// TwinCAT 3 PLC project XtsTransport
// Title: XTS Transport
// Author: D.Hauer
// ProjectVersion: 3.2.8
// Description: basic functionblocks for building XTS transport
// ProgramVersion: 3.1.4026.19
// libraries:
//   Tc2_Math, * (Beckhoff Automation GmbH)
//   Tc2_MC2, * (Beckhoff Automation GmbH)
//   Tc2_Standard, * (Beckhoff Automation GmbH)
//   Tc2_System, * (Beckhoff Automation GmbH)
//   Tc2_Utilities, * (Beckhoff Automation GmbH)
//   Tc3_McCollisionAvoidance, * (Beckhoff Automation GmbH)
//   Tc3_McCoordinatedMotion, * (Beckhoff Automation GmbH)
//   Tc3_Module, * (Beckhoff Automation GmbH)
//   Tc3_XTS_Utility, * (Beckhoff Automation GmbH)
//   VisuDialogs, * (System)
// project tree:
//   / GlobalTextList.TcGTLO (not stored), MAIN.TcPOU, PlcTask.TcTTO
//   MAPPING/ MAPPING_in.TcPOU, MAPPING_out.TcPOU
//   MAPPING/_types/ U_GEAR_DATA.TcDUT (not stored), U_MOVER_CTRL.TcDUT (not stored), U_MOVER_INFO.TcDUT (not stored), U_MOVER_STATE.TcDUT (not stored), U_MOVE_DATA.TcDUT (not stored), U_XTS_STATION_CTRL.TcDUT (not stored), U_XTS_STATION_STATE.TcDUT (not stored), U_XTS_TRANSPORT_CTRL.TcDUT (not stored), U_XTS_TRANSPORT_STATE.TcDUT (not stored)
//   MSG/ fb_LocalTime.TcPOU (not stored), f_MessageSet.TcPOU, GVL_MSG.TcGVL, MessageData.TcPOU (not stored), T_MESSAGE_LIST.TcVIS
//   MSG/types/ e_Device.TcDUT (not stored), E_MessageType.TcDUT (not stored), E_MESSAGE_STATE.TcDUT, e_Subdevice.TcDUT (not stored), ST_Message.TcDUT (not stored), TL_E_MESSAGETYPE.TcTLO
//   XTS/CaGroup/ FB_CaGroup.TcPOU, I_XtsTransport_CaGroup.TcIO (not stored)
//   XTS/CaGroup/types/ E_CA_GROUP_STATE.TcDUT (not stored), E_GROUP_CHECK.TcDUT (not stored), ST_GROUP_INFO.TcDUT (not stored)
//   XTS/ GVL_XTS.TcGVL (not stored), XTS_Parameter.TcGVL
//   XTS/Mover/ fb_Mover.TcPOU, fb_MoverCtrl.TcPOU (not stored), I_XtsTransport_Mover.TcIO
//   XTS/Mover/types/ E_MOVER_CTRL.TcDUT (not stored), E_MOVER_STATE.TcDUT, ST_GEAR_DATA.TcDUT, ST_MOVER_CTRL.TcDUT (not stored), ST_MOVER_INFO.TcDUT (not stored), ST_MOVER_STATE.TcDUT (not stored), ST_MOVE_DATA.TcDUT (not stored)
//   XTS/XtsStation/ fb_Station.TcPOU, I_XtsTransport_Station.TcIO (not stored)
//   XTS/XtsStation/_types/ E_STATION_CTRL.TcDUT (not stored), E_STATION_STATE.TcDUT, fb_Station_LinkedListCtrl.TcPOU, I_Station_LinkedList.TcIO (not stored), ST_STATION_CTRL.TcDUT (not stored), ST_STATION_LIST_RESULT.TcDUT (not stored), ST_STATION_MOVER_DATA.TcDUT (not stored), ST_STATION_PARAMETER.TcDUT (not stored), ST_STATION_STATE.TcDUT, T_NEST_OFFSET.TcDUT (not stored)
//   XTS/Xpu/ fb_Xpu.TcPOU, fb_XpuCtrl.TcPOU (not stored)
//   XTS/Xpu/types/ E_XPU_CHECK.TcDUT, E_XPU_CTRL.TcDUT (not stored), E_XPU_INIT.TcDUT (not stored), E_XPU_STATE.TcDUT (not stored), ST_XPU_CTRL.TcDUT (not stored), ST_XPU_INFO.TcDUT (not stored), ST_XPU_STATE.TcDUT (not stored)
//   XTS/XtsTransportUnit/ fb_TransportUnit.TcPOU
//   XTS/XtsTransportUnit/types/ E_XTS_TRANSPORT_CHECK.TcDUT (not stored), E_XTS_TRANSPORT_CTRL.TcDUT (not stored), E_XTS_TRANSPORT_STATE.TcDUT (not stored), ST_XTS_TRANSPORT_CTRL.TcDUT (not stored), ST_XTS_TRANSPORT_STATE.TcDUT (not stored)
//   XTS/_types/ E_PROGRESS.TcDUT (not stored), f_GetProgress.TcPOU (not stored), f_GetState.TcPOU (not stored)

CONFIGURATION XtsTransport
    RESOURCE PLC ON TwinCAT3
        TASK PlcTask(INTERVAL := T#2ms, PRIORITY := 15);
        PROGRAM MAPPING_in WITH PlcTask : MAPPING_in;
        PROGRAM MAIN WITH PlcTask : MAIN;
        PROGRAM MAPPING_out WITH PlcTask : MAPPING_out;
    END_RESOURCE
END_CONFIGURATION

// ---- MSG/types/E_MESSAGE_STATE.TcDUT
{attribute 'strict'}
TYPE E_MESSAGE_STATE :
(
  MSG_INVALID_POINTERS  := -1,
	MSG_NULL,
  MSG_INIT,
  MSG_ROOT              := 10,
  MSG_ROOT_CREATE,
  MSG_ROOT_CREATE_BUSY,
  MSG_FOLDER,
  MSG_FOLDER_CREATE,
  MSG_FOLDER_CREATE_BUSY,
  MSG_FILE_CREATE_DONE,
  MSG_LINE_START        := 100,
  MSG_LINE_BUILD,
  MSG_LINE_CHECK,
  MSG_WRITE_FILE_BUSY  := 200,
  MSG_WRITE_FILE_END,
  MSG_WRITE_FILE_DONE   := 1000
)DINT;
END_TYPE

// ---- XTS/Mover/types/E_MOVER_STATE.TcDUT
{attribute 'qualified_only'}
{attribute 'to_string'}
TYPE E_MOVER_STATE :
(
  MOVER_NULL,               // initial value at startup, used for change of order or retrigger
  MOVER_ENABLE,             // sets MC_Power.Enable
  MOVER_DISABLE,            // removes MC_Power.Enable
  MOVER_MOVE_TO_POS,        // modulo absolute positioning with MC_MoveAbsolute, InTargetPosition check
  MOVER_MOVE_TO_POS_CA,     // modulo absolute positioning with MC_MoveAbsoluteCA, InTargetPosition check
  MOVER_SEND_TO_POS_CA,     // modulo absolute positioning with MC_MoveAbsoluteCA, done after moving ReleaseDistance
  MOVER_HALT,               // halts mover; by use of MC_Halt mover is set passive in CA group
  MOVER_GEAR_IN,            // GearIn for mover in standstill

  MOVER_GEAR_IN_POS_CA,     // GearInPosCA of mover; when FB_GearInPosCa is InSync --> order is done; check SyncDistance yourself and release mover with e_mover_order.mover_SendToPos
  MOVER_GEAR_OUT,           // gear out for mover
  MOVER_RESET               // MC_RESET for mover
)UINT;
END_TYPE

// ---- XTS/Mover/types/ST_GEAR_DATA.TcDUT
{attribute 'pack_mode' := '2'}
TYPE ST_GEAR_DATA :
STRUCT
  rDeltaToMasterPos       : LREAL;
  rModuloSyncPosSlave     : LREAL;
  rMasterStartDistance    : LREAL;
  rGearNumerator          : LREAL;
  iGearDenumerator        : USINT  := 1;
END_STRUCT
END_TYPE

// ---- XTS/XtsStation/_types/E_STATION_STATE.TcDUT
{attribute 'qualified_only'}
{attribute 'to_string'}

TYPE E_STATION_STATE :
(
	STATION_NO_INIT,                // startup state after power on, first cycle Init of station, switches to INIT when done

  STATION_INIT,                   // CONTINUE to DISABLE
                                  // State.MoverId deleted

  STATION_DISABLE         := 10,  // + CTRL.STATION_ENABLE  --> CONTINUE to DETECT_MOVER 
                                  // station is empty, no mover is handled, check enable from ctrl

  STATION_ENABLE,                 // init of work vars, check enable from ctrl

  STATION_DETECT_MOVER,           // (QueueCount > 0)       --> CONTINUE to MOVER_ENTER

  STATION_MOVER_ENTER     := 20,  // + CTRL.MOVER_ENTER     --> CONTINUE to PROCESS_START
                                  // + CTRL.MOVER_SEND      --> CONTINUE to MOVER_OUT
                                  // mover asking for entry

  STATION_MOVER_IN_TARGET,        // (MoveToPos==TRUE)      --> CONTINUE to PROCESS_START
                                  // mover is moving to PosWait + PosStop[_nNest]

  STATION_PROCESS_START   := 30,  // + CTRL.PROCESS_START   --> CONTINUE to PROCESS_START
                                  // + CTRL.PROCESS_DONE    --> CONTINUE to CHECK
                                  // wait until process started

  STATION_PROCESS_DONE,           // + CTRL.PROCESS_DONE    --> CONTINUE to CHECK
                                  // wait until process done

  STATION_CHECK           := 40,  // check for next nest in mask, 
                                  // (mask<>0) --> CHECK_NEST
                                  // (mask==0) --> MOVER_OUT

  STATION_CHECK_NEST,             // + CTRL.MOVER_ENTER     --> CONTINUE to MOVER_IN_TARGET
                                  // get next nest position








  STATION_MOVER_OUT       := 50,          // + CTRL.MOVER_OUT       --> CONTINUE to MOVER_RELEASE
                                          // mover asking to leave

  STATION_MOVER_RELEASE,                  // (MoverSendToPos==TRUE) --> CONTINUE to MOVER_GONE
                                          // mover is released + check if release distance is passed

  STATION_MOVER_WRITE_TARGET,             // worker state to write mover ticket








  STATION_MOVER_GONE      := 60,          // + CTRL.MOVER_GONE      --> CONTINUE to INIT
                                          // mover out of station, enter mover in target station list


  STATION_ERROR_NULL      := 127,
  STATION_ERROR_LIST_GET_HEAD_FAULT,      // fatal error in linked list, must never occurr, must be debugged
  STATION_ERROR_LIST_REMOVE_HEAD_FAULT,   // fatal error in linked list, must never occurr, must be debugged
  STATION_ERROR_LIST_ADD_TAIL_FAULT,      // fatal error in linked list, must never occurr, must be debugged

  STATION_ERROR_LIST_STATION_ID_WRONG,    // ticket data in Queue contains wrong Station Id, can be overruled by ctrl

  STATION_ERROR_LIST_MOVER_ID_INVALID,    // fatal error in ticket data, MoverId is out of range, must be fixed by ctrl, must be debugged

  STATION_ERROR_INFEED_ERROR,             // motion error during movement, retry must be triggered by ctrl
  STATION_ERROR_OUTFEED_ERROR,            // motion error during movement, retry by ctrl OR leave by ctrl

  STATION_ERROR_OUTFEED_TARGET_INVALID,   // ticket data for nTargetStation is not plausible, can be fixed by ctrl

  STATION_ERROR_FATAL     := 255          // the thing that must not be, all fatal errors end up here
)USINT;
END_TYPE

// ---- XTS/XtsStation/_types/ST_STATION_STATE.TcDUT
{attribute 'pack_mode' := '2'}
TYPE ST_STATION_STATE :
STRUCT
  eState          : E_STATION_STATE;
  {attribute 'displaymode':='bin'}
  nMask           : BYTE;
  nMoverId        : USINT;
  rMoverModPos    : LREAL;            // modulo position of detected mover
  nQueue          : USINT;            // queue count for station
END_STRUCT
END_TYPE

// ---- XTS/Xpu/types/E_XPU_CHECK.TcDUT
{attribute 'qualified_only'}
{attribute 'to_string'}
TYPE E_XPU_CHECK :
(
  INIT_CHECK,
  INIT_CHECK_ERROR,
  START_CHECK,
  XPU_INSTANCE_NULL,
  XPU_RAIL_LENGTH,
  GROUP_RAIL_LENGTH,
  RAIL_LENGTH_COMPARE,
  GROUP_NOT_CONFIGURED,
  GROUP_OID_MISMATCH,

  MOVER_COUNT             := 10,
  MOVER_COUNT_ZERO,
  MOVER_COUNT_NOT_EQUAL,

  PROCESSING_UNIT_POSITIONS_VALID         := 20,
  PROCESSING_UNIT_GET_DATA_EXCEED,

  MOVER_ID_STANDARD       := 30,
  MOVER_ID_SIMULATION,
  MOVER_ID_DETECTION_MODE,
  MOVER_ID_DETECTION_VALID,
  MOVER_ID_DETECTION_DC_LINK,
  MOVER_ID_DETECTION_BUSY,
  MOVER_ID_DETECTION_IDLE,
  MOVER_ID_DETECTION_STATE,
  MOVER_ID_MULTIPLE_NOT_SUPPORTED,

  POINTER_CHECK           := 90,
  POINTER_NULL_CTRL,
  POINTER_NULL_STATE
)UINT;
END_TYPE

// ---- MSG/GVL_MSG.TcGVL
{attribute 'qualified_only'}
VAR_GLOBAL CONSTANT
  //-----------------------------------------------------------------------------
  // file paths for message system
  //  - compiler define option WIN switches to Windows file paths
  //-----------------------------------------------------------------------------
{IF defined (WIN)}
  {info 'WIN folders'}
  LOG_DIR               : STRING  := 'C:\TwinCAT\#MsgFiles\';
  CONFIG_DIR            : STRING  := 'C:\TwinCAT\XPU_PLC_StationConfig\';
{ELSE}
  {info 'BSD folders'}
  LOG_DIR               : STRING  := '/usr/local/etc/TwinCAT/#MsgFiles/';
  CONFIG_DIR            : STRING  := '/usr/local/etc/TwinCAT/XPU_PLC_StationConfig/';
{END_IF}

  LOG_FILE              : STRING  := 'MSG_XtsTransport_';
  CONFIG_FILE           : STRING  := 'Config_XPU_'; // OTCID of fb_Environment is added to name on writing

  MAX_MESSAGE           : UINT    := 200; // max entry in message list
END_VAR
VAR_GLOBAL
  Messages                        : ARRAY[1..MAX_MESSAGE] OF ST_Message;
  MessageIndex                    : UINT := 0; // message index
  MessageError                    : UINT := 0; // error counter

  fbLocalTime                     : fb_LocalTime;
  dtLocalTime                     : DT;
  sLocalTime                      : STRING;

  MessageLevelXpu            AT %I*     : E_MessageType;
  MessageLevelGroup          AT %I*     : E_MessageType;
  MessageLevelTransport      AT %I*     : E_MessageType;
  MessageLevelStations       AT %I*     : ARRAY[1..MAX_STATION] OF E_MessageType;
  MessageLevelMovers                    : ARRAY[1..MAX_MOVER]   OF E_MessageType;


{IF defined (TEST)}
  {info 'TEST logging enabled'}
  MessageLevel                    : E_MessageType := eMessageVerbose; // a lot of messages
{ELSE}
  MessageLevel                    : E_MessageType := eMessageError;   // only errors are written into list 
{END_IF}

END_VAR

// ---- XTS/XTS_Parameter.TcGVL
//{attribute 'qualified_only'}
VAR_GLOBAL CONSTANT
// HAUD 2025 08 09
//
//    XTS_TRANSPORT_LAYER project
//    
//    MIT License
//    
//    Copyright (c) 2025 HAUD
//    
//    Permission is hereby granted, free of charge, to any person obtaining a copy
//    of this software and associated documentation files (the "Software"), to deal
//    in the Software without restriction, including without limitation the rights
//    to use, copy, modify, merge, publish, distribute, sublicense, and/or sell
//    copies of the Software, and to permit persons to whom the Software is
//    furnished to do so, subject to the following conditions:
//    
//    The above copyright notice and this permission notice shall be included in all
//    copies or substantial portions of the Software.
//    
//    THE SOFTWARE IS PROVIDED "AS IS", WITHOUT WARRANTY OF ANY KIND, EXPRESS OR
//    IMPLIED, INCLUDING BUT NOT LIMITED TO THE WARRANTIES OF MERCHANTABILITY,
//    FITNESS FOR A PARTICULAR PURPOSE AND NONINFRINGEMENT. IN NO EVENT SHALL THE
//    AUTHORS OR COPYRIGHT HOLDERS BE LIABLE FOR ANY CLAIM, DAMAGES OR OTHER
//    LIABILITY, WHETHER IN AN ACTION OF CONTRACT, TORT OR OTHERWISE, ARISING FROM,
//    OUT OF OR IN CONNECTION WITH THE SOFTWARE OR THE USE OR OTHER DEALINGS IN THE
//    SOFTWARE.

  Version             : STRING  := '4.00.11';

  MAX_MOVER           : UINT    := TO_UINT(Tc3_XTS_Utility.TcIoXtsEnvironmentParameterList.MaxXtsMoversPerXpu);
  MAX_MODULE          : UINT    := TO_UINT(Tc3_XTS_Utility.TcIoXtsEnvironmentParameterList.MaxModulesPerPart);
  MAX_PART            : UINT    := TO_UINT(Tc3_XTS_Utility.TcIoXtsEnvironmentParameterList.MaxXtsPartsPerXpu);
  MAX_TRACK           : UINT    := TO_UINT(Tc3_XTS_Utility.TcIoXtsEnvironmentParameterList.MaxXtsTracksPerXpu);
  MAX_GROUP           : UINT    := TO_UINT(Tc3_XTS_Utility.TcIoXtsEnvironmentParameterList.MaxXtsCaGroup);

  MAX_INFO_SERVER     : UINT    := TO_UINT(Tc3_XTS_Utility.TcIoXtsEnvironmentParameterList.MaxXtsInfoServer);
  MAX_INFO_STATION    : UINT    := TO_UINT(Tc3_XTS_Utility.TcIoXtsEnvironmentParameterList.MaxXtsInfoStation);
  MAX_INFO_STOP_POS   : UINT    := TO_UINT(Tc3_XTS_Utility.TcIoXtsEnvironmentParameterList.MaxXtsStopPositionsPerStation);

  MAX_PARAMETER_SET   : UINT    := TO_UINT(Tc3_XTS_Utility.TcIoXtsEnvironmentParameterList.MaxXtsParameterSet);

  MAX_NCT_BASE_UNIT   : UINT    := TO_UINT(Tc3_XTS_Utility.TcIoXtsEnvironmentParameterList.MaxXtsNctBaseUnitInterfaces);

  MAX_STATION         : UINT    := 5;

  MAX_STATION_NEST    : UINT    := TO_UINT(SIZEOF(ST_STATION_STATE.nMask)*8);
  // MAX_LIST_NODES      : UINT    := MAX_MOVER;
  MAX_LIST_NODES      : UINT    := 24; // visualization can not handle access to MAX_MOVER
  MAX_MASTER          : UINT    := 1;
END_VAR

// ---- XTS/Mover/I_XtsTransport_Mover.TcIO
INTERFACE I_XtsTransport_Mover

METHOD Disable : E_PROGRESS
VAR_INPUT
  Execute             : BOOL;
END_VAR
END_METHOD

METHOD Enable : E_PROGRESS
VAR_INPUT
  Execute             : BOOL;
END_VAR
END_METHOD

METHOD GearIn : E_PROGRESS;
VAR_INPUT
  Execute             : BOOL;
  stMoveData          : ST_MOVE_DATA;
  stGearData          : ST_GEAR_DATA;
END_VAR
END_METHOD

METHOD GearInPosCa : E_PROGRESS
VAR_INPUT
  Execute             : BOOL;
  stMoveData          : ST_MOVE_DATA;
  stGearData          : ST_GEAR_DATA;  
END_VAR
END_METHOD

METHOD GearOut : E_PROGRESS
VAR_INPUT
  Execute             : BOOL;
END_VAR
END_METHOD

METHOD Halt : E_PROGRESS
VAR_INPUT
  Execute             : BOOL;
  stMoveData          : ST_MOVE_DATA;
END_VAR
END_METHOD

METHOD HaltCa : E_PROGRESS
VAR_INPUT
  Execute             : BOOL;
  stMoveData          : ST_MOVE_DATA;
END_VAR
END_METHOD

PROPERTY MessageLevel : e_messagetype
SET
END_SET
END_PROPERTY

PROPERTY ModuloTurn : dint
GET
END_GET
END_PROPERTY

METHOD MoveToPos : E_PROGRESS
VAR_INPUT
  Execute             : BOOL;
  stMoveData          : ST_MOVE_DATA;
END_VAR
END_METHOD

METHOD MoveToPosCa : E_PROGRESS
VAR_INPUT
  Execute             : BOOL;
  stMoveData          : ST_MOVE_DATA;
END_VAR
END_METHOD

PROPERTY RailLength : LREAL
GET
END_GET
SET
END_SET
END_PROPERTY

METHOD Reset : E_PROGRESS
VAR_INPUT
  Execute             : BOOL;
END_VAR
END_METHOD

METHOD SendToAbsPosCa : E_PROGRESS
VAR_INPUT
  Execute             : BOOL;
  stMoveData          : ST_MOVE_DATA;
END_VAR
END_METHOD

METHOD SendToModuloPosCa : E_PROGRESS
VAR_INPUT
  Execute             : BOOL;
  stMoveData          : ST_MOVE_DATA;
END_VAR
END_METHOD

METHOD Stop : E_PROGRESS
VAR_INPUT
  Execute             : BOOL;
  stMoveData          : ST_MOVE_DATA;
END_VAR
END_METHOD

END_INTERFACE

// ---- MAPPING/MAPPING_in.TcPOU
PROGRAM MAPPING_in
VAR CONSTANT
{IF defined (MOVER_MAP)}
  {info 'MAPPING_in - MOVER_MAPPING active'}
  bBypassMappingMover       : BOOL  := FALSE;
{ELSE}
  bBypassMappingMover       : BOOL  := TRUE;
{END_IF}
{IF defined (STATION_MAP)}
  {info 'MAPPING_in - STATION_MAPPING active'}
  bBypassMappingStation     : BOOL  := FALSE;
{ELSE}
  bBypassMappingStation     : BOOL  := TRUE;
{END_IF}
END_VAR
VAR
  bBypassInput      : BOOL;
  sMapping          : STRING;

  bFirstCycle       : BOOL := TRUE;
{IF defined (MOVER_MAP)}
  MoverCtrl         : U_MOVER_CTRL;
  MoveData          : U_MOVE_DATA;
  GearData          : U_GEAR_DATA;

{ELSE}
  MoverCtrl         : BYTE;
  MoveData          : BYTE;
  GearData          : BYTE;
{END_IF}
{IF defined (STATION_MAP)}
  StationControl    : U_XTS_STATION_CTRL;
{ELSE}
  StationControl    : BYTE;
{END_IF}

  TransportControl  : U_XTS_TRANSPORT_CTRL;

  szGearData,
  szMoveData,
  szMoverCtrl         : ARRAY[1..2] OF UDINT;

  szStationCtrl       : ARRAY[1..2] OF UDINT;

  szTransportCtrl     : ARRAY[1..2] OF UDINT;
END_VAR


IF (bFirstCycle)
THEN
  bFirstCycle             := FALSE;

  szMoverCtrl[1]          := SIZEOF(MoverCtrl);
  szMoverCtrl[2]          := SIZEOF(GVL_XTS.MoverCtrl);
  
  szMoveData [1]          := SIZEOF(MoveData);
  szMoveData [2]          := SIZEOF(GVL_XTS.MoveData);
  
  szGearData [1]          := SIZEOF(GearData);
  szGearData [2]          := SIZEOF(GVL_XTS.GearData);
  
  szStationCtrl[1]        := SIZEOF(StationControl);
  szStationCtrl[2]        := SIZEOF(GVL_XTS.StationCtrl);

  szTransportCtrl[1]      := SIZEOF(TransportControl);
  szTransportCtrl[2]      := SIZEOF(GVL_XTS.XtsTransportCtrl);
END_IF

IF (bBypassInput) 
THEN 
  sMapping  := 'NO_MAPPING_ACTIVE';
  RETURN;
ELSE
  sMapping  := 'MAPPING_ACTIVE';
END_IF

IF NOT bBypassMappingMover
THEN
  memcpy(ADR(GVL_XTS.MoverCtrl),        ADR(MoverCtrl),         SIZEOF(MoverCtrl));
  memcpy(ADR(GVL_XTS.MoveData),         ADR(MoveData),          SIZEOF(MoveData));
  memcpy(ADR(GVL_XTS.GearData),         ADR(GearData),          SIZEOF(GearData));
END_IF

IF NOT bBypassMappingStation
THEN
  memcpy(ADR(GVL_XTS.StationCtrl),      ADR(StationControl),    SIZEOF(StationControl));
END_IF

  memcpy(ADR(GVL_XTS.XtsTransportCtrl), ADR(TransportControl),     SIZEOF(TransportControl));

END_PROGRAM

// ---- MAIN.TcPOU
//---------------------------------------------------------------------------------------------------------------
//
//  HAUD 2024.03.18
//
//  - XTS_TRANSPORT_LAYER
//  - transport layer members:
//    - CaGroup
//      - access to Group functions
//
//    - Mover
//      - access to MC and CA motion functions
//
//    - Xpu (ProcessingUnit)
//      - access to TcCOM Objects in Environment
//
//    - Transport Control Unit
//      - coordinates members to get XTS in defined states
//
//    - Xts Stations
//      - handshakes with extern control for mover transport
//
//  - global datafields for mrmbers in GVL_XTS namespace
//  - global interface datafields for use in members
//  - structures are assigned by reference for every member
//
//---------------------------------------------------------------------------------------------------------------
// HAUD 2024 05 29
//
//    XTS_TRANSPORT_LAYER project
//    
//    MIT License
//    
//    Copyright (c) 2024 HAUD
//    
//    Permission is hereby granted, free of charge, to any person obtaining a copy
//    of this software and associated documentation files (the "Software"), to deal
//    in the Software without restriction, including without limitation the rights
//    to use, copy, modify, merge, publish, distribute, sublicense, and/or sell
//    copies of the Software, and to permit persons to whom the Software is
//    furnished to do so, subject to the following conditions:
//    
//    The above copyright notice and this permission notice shall be included in all
//    copies or substantial portions of the Software.
//    
//    THE SOFTWARE IS PROVIDED "AS IS", WITHOUT WARRANTY OF ANY KIND, EXPRESS OR
//    IMPLIED, INCLUDING BUT NOT LIMITED TO THE WARRANTIES OF MERCHANTABILITY,
//    FITNESS FOR A PARTICULAR PURPOSE AND NONINFRINGEMENT. IN NO EVENT SHALL THE
//    AUTHORS OR COPYRIGHT HOLDERS BE LIABLE FOR ANY CLAIM, DAMAGES OR OTHER
//    LIABILITY, WHETHER IN AN ACTION OF CONTRACT, TORT OR OTHERWISE, ARISING FROM,
//    OUT OF OR IN CONNECTION WITH THE SOFTWARE OR THE USE OR OTHER DEALINGS IN THE
//    SOFTWARE.
//---------------------------------------------------------------------------------------------------------------
PROGRAM MAIN
VAR
	bInit 				  : BOOL;
  eInit   AT%Q*   : E_PROGRESS;

  nStation,
	nMover,
  nMoverSelected,
  nStationSelected,
  nStationParameter   : UINT;

  sStationText        : STRING(30);

  eTransportState     : E_XTS_TRANSPORT_STATE;
  eTransportResult    : E_PROGRESS;

  eXpuState           : E_XPU_STATE;
  eXpuResult          : E_PROGRESS;
  eXpuCheck           : E_XPU_CHECK;

  eMoverState         : E_MOVER_STATE;
  eMoverResult        : E_PROGRESS;

  sCaGroupState,
  sTransportState,
  sTransportCheck,
  sTransportResult,
  sXpuState,
  sXpuResult,
  sXpuCheck,
  sXpuOpMode,
  sXpuMoverdetectionMode,
  sXpuMoverAssignement,
  sMoverState,
  sMoverResult,
  sStationState,
  sStationStateMask,
  sStationCtrlMask        : STRING;

  bStationEnable,
  bStationEnter,
  bStationStart,
  bStationDone,
  bStationOut,
  bStationGone            : BOOL;

  tStationSelectedQueue   : ARRAY[1..MAX_LIST_NODES] OF ST_STATION_MOVER_DATA;

  tonWriteLog             : Tc2_Standard.TON;
  tWriteLog               : TIME := T#5S;
END_VAR

//############################################################################
// Local time; used for timestamps
//############################################################################
GVL_MSG.fbLocalTime(
                    sLocalTime          => GVL_MSG.sLocalTime, 
                    dtLocalTime         => GVL_MSG.dtLocalTime);
//############################################################################

//############################################################################
// 	example for init sequence
//############################################################################	
IF NOT bInit
THEN
  CASE eInit
  OF
    E_PROGRESS.PROGRESS_INVALID,
    E_PROGRESS.PROGRESS_DONE:         // clear command interface
      eInit                                   := E_PROGRESS.PROGRESS_BUSY;
      GVL_XTS.XpuCtrl.Cmd                     := E_XPU_CTRL.XTS_CMD_NULL;


    E_PROGRESS.PROGRESS_BUSY:         // init Xpu, ProcessingUnit, MotorModules
      eInit                                   := E_PROGRESS.PROGRESS_PREPARE;
      GVL_XTS.XpuCtrl.Cmd                     := E_XPU_CTRL.XTS_CMD_INIT;

    E_PROGRESS.PROGRESS_PREPARE:      // wait for init to be done
      IF (GVL_XTS.XpuState.State      = E_XPU_STATE.XTS_INIT + E_PROGRESS.PROGRESS_DONE)
      THEN
        eInit                                 := E_PROGRESS.PROGRESS_STARTUP;
        GVL_XTS.XpuCtrl.Cmd                   := E_XPU_CTRL.XTS_IDLE;
      END_IF

    E_PROGRESS.PROGRESS_STARTUP:      // assign mover interfaces
      eInit                                   := E_PROGRESS.PROGRESS_CHECK;
      FOR nMover := 1 TO MAX_MOVER
      DO
        GVL_XTS.MoverItf[nMover]              := GVL_XTS.Mover[nMover];
      END_FOR

    E_PROGRESS.PROGRESS_CHECK:        // assign CaGroup interface
      eInit                                   := E_PROGRESS.PROGRESS_OCCUPIED;
      GVL_XTS.CaGroupItf                      := GVL_XTS.CaGroup;

    E_PROGRESS.PROGRESS_OCCUPIED:     // StartStation for XtsTransportCtrl.Cmd := E_XTS_TRANSPORT_CTRL.CMD_TRANSPORT_START;
      eInit                                   := E_PROGRESS.PROGRESS_WORKING;
      // where to start?
      GVL_XTS.XtsTransport.StationStartIndex  := 1;

      // Start Position parameters
      GVL_XTS.StationStart.rPosWait           :=     10.0;
      GVL_XTS.StationStart.rGap               :=    150.0;
      GVL_XTS.StationStart.rVelo              :=   1250.0;
      GVL_XTS.StationStart.rAccDec            :=  12000.0;
      GVL_XTS.StationStart.rJerk              := 400000.0;

    E_PROGRESS.PROGRESS_WORKING:
      // hard coded XTS Station parameter are here:
      StationParameterInit();

      // initialization of XtsTransport is done here:
      bInit                                   := TRUE;
      eInit                                   := E_PROGRESS.PROGRESS_DONE;
  END_CASE
END_IF

//############################################################################
// 	XTS Transport Unit
//############################################################################
//  - main control function block for transport layer
//  - requires access to member controls
//    - Xpu
//    - CaGroup
//    - Mover
//    - Station Control
//    - Station LinkedList Interface
//############################################################################
//
// cyclic call
GVL_XTS.XtsTransport();

GVL_XTS.XtsTransport.MessageLevel       := GVL_MSG.MessageLevelTransport;

// main control
GVL_XTS.XtsTransport.Ctrl               REF= GVL_XTS.XtsTransportCtrl;   // main control
GVL_XTS.XtsTransport.State              REF= GVL_XTS.XtsTransportState;  // main state
                                        
// member controls                      
GVL_XTS.XtsTransport.XpuCtrl            REF= GVL_XTS.XpuCtrl;
GVL_XTS.XtsTransport.XpuState           REF= GVL_XTS.XpuState;
GVL_XTS.XtsTransport.XpuInfo            REF= GVL_XTS.XpuInfo;
                                        
GVL_XTS.XtsTransport.GroupItf           :=   GVL_XTS.CaGroupItf;
GVL_XTS.XtsTransport.GroupInfo          REF= GVL_XTS.CaGroupInfo;
                                        
GVL_XTS.XtsTransport.MoverItf           REF= GVL_XTS.MoverItf;
GVL_XTS.XtsTransport.MoverInfo          REF= GVL_XTS.MoverInfo;
GVL_XTS.XtsTransport.MoverLastPosition  REF= GVL_XTS.LastPosition;
GVL_XTS.XtsTransport.MoverLastGap       REF= GVL_XTS.LastGap;
                                        
GVL_XTS.XtsTransport.StationStart       REF= GVL_XTS.StationStart;      // start position for E_XTS_TRANSPORT_CTRL.CMD_TRANSPORT_START
GVL_XTS.XtsTransport.StationCtrlItf     REF= GVL_XTS.StationCtrlItf;    // station interfaces are required for accessing station methods
GVL_XTS.XtsTransport.StationListsItf    REF= GVL_XTS.StationListItf;    // list interface is required for access to linked list methods
GVL_XTS.XtsTransport.StationControl     REF= GVL_XTS.StationCtrl;
GVL_XTS.XtsTransport.StationState       REF= GVL_XTS.StationState;
//############################################################################



//############################################################################
// 	XTS Stations
//############################################################################	
FOR nStation := 1 TO MAX_STATION
DO
  GVL_XTS.Station[nStation].MessageLevel:= GVL_MSG.MessageLevelStations[nStation];

  GVL_XTS.Station[nStation].StationId   := nStation;
  GVL_XTS.Station[nStation].MessageLevel:= GVL_MSG.MessageLevelStations[nStation];

  GVL_XTS.StationListItf[nStation]      := GVL_XTS.StationList[nStation];   // interfaces for list methods
  GVL_XTS.StationCtrlItf[nStation]      := GVL_XTS.Station[nStation];       // interfaces for station methods

  GVL_XTS.Station[nStation].Ctrl        REF= GVL_XTS.StationCtrl;           // station ctrl from extern
  GVL_XTS.Station[nStation].State       REF= GVL_XTS.StationState;          // station state to extern

  GVL_XTS.Station[nStation].ItfStations REF= GVL_XTS.StationListItf;        // give every station all list interfaces for writing mover tickets
  GVL_XTS.Station[nStation].ItfMover    REF= GVL_XTS.MoverItf;              // give every station all mover interfaces for movement in / out of station
  GVL_XTS.Station[nStation].Mover       REF= GVL_XTS.AxisRefMover;          // AXIS_REF to read infos from
  GVL_XTS.Station[nStation].MoverOffset REF= GVL_XTS.PositionOffset;        // static offsets for all stations, all movers, all stop positions


  GVL_XTS.Station[nStation].StationParameter  REF= GVL_XTS.StationParameter;// give every station all station parameters for sending to WaitPos of target station

  // cyclic call
  GVL_XTS.Station[nStation].Cycle();                                        // cycle for handshaking with extern

  // Queue data for each station
  GVL_XTS.StationQueue[nStation]        := GVL_XTS.StationListItf[nStation].Data;
END_FOR
//############################################################################



//############################################################################
// 	XPU environment
//############################################################################	
GVL_XTS.Xpu.XpuInstance               :=   1;
GVL_XTS.Xpu.MessageLevel              :=   GVL_MSG.MessageLevelXpu;

GVL_XTS.Xpu.Ctrl                      REF= GVL_XTS.XpuCtrl;
GVL_XTS.Xpu.State                     REF= GVL_XTS.XpuState;
GVL_XTS.Xpu.XpuModuleInfoData         REF= GVL_XTS.XpuModules;

GVL_XTS.Xpu.CaGroupOID                :=   GVL_XTS.CaGroup.GroupInfo.CaGroupOID;

// cyclic call
GVL_XTS.Xpu();
GVL_XTS.XpuInfo                       :=   GVL_XTS.Xpu.XpuInfo;
//############################################################################


//############################################################################	
// 	CA-Group Class
//############################################################################	
// assignment
GVL_XTS.CaGroup.MessageLevel          := GVL_MSG.MessageLevelGroup;

GVL_XTS.CaGroup.AxisRef               REF= GVL_XTS.AxisRefMover;
// Interface to Mover methods
GVL_XTS.CaGroup.MoverItf              REF= GVL_XTS.MoverItf; 

GVL_XTS.CaGroup.GroupRef              REF= GVL_XTS.CaGroupRef;

// cyclic call
GVL_XTS.CaGroup.InfoCycle(TRUE); // read group status

// InfoData from group
GVL_XTS.CaGroupInfo                   :=   GVL_XTS.CaGroup.GroupInfo;

// Interface of CaGroup
GVL_XTS.CaGroupItf                    :=   GVL_XTS.CaGroup;
//############################################################################


//############################################################################
// Mover Class	
//############################################################################	
FOR nMover := 1 TO MAX_MOVER
DO
  GVL_XTS.Mover[nMover].MessageLevel  := GVL_MSG.MessageLevelMovers[nMover];

  GVL_XTS.Mover[nMover].MoverId       :=   nMover;
  GVL_XTS.Mover[nMover].RailLength    :=   GVL_XTS.Xpu.RailLength;  // mover needs RailLength, in order to calc absolute position from modulo input
  GVL_XTS.Mover[nMover].MessageLevel  :=   GVL_MSG.MessageLevelMovers[nMover];

  GVL_XTS.Mover[nMover].Ctrl          REF= GVL_XTS.MoverCtrl;       // mover control from extern
  GVL_XTS.Mover[nMover].State         REF= GVL_XTS.MoverState;      // mover state to extern

  GVL_XTS.Mover[nMover].MoveData      REF= GVL_XTS.MoveData;        // dyn constraints for extern to write
  GVL_XTS.Mover[nMover].GearData      REF= GVL_XTS.GearData;        // GearIn/GearInPosCa data fro extern to write

  // assignment	
  GVL_XTS.Mover[nMover].Mover         REF= GVL_XTS.AxisRefMover[nMover];  // axis reference to Mover function block
  GVL_XTS.Mover[nMover].LastGap       REF= GVL_XTS.LastGap[nMover];       // reference to last used gap value datafield
  GVL_XTS.Mover[nMover].LastPosition  REF= GVL_XTS.LastPosition[nMover];  // reference to last position datafield

  GVL_XTS.Mover[nMover].MoverInfo		  REF= GVL_XTS.MoverInfo[nMover];     // refernence to mover info data (ActPos, SetPos, ...)

  GVL_XTS.MoverItf[nMover]            :=   GVL_XTS.Mover[nMover];

  // cyclic call
  GVL_XTS.Mover[nMover].Cycle();  // call AXIS_REF()
  GVL_XTS.Mover[nMover]();        // call Ctrl/State
END_FOR


//############################################################################


//############################################################################
// /logging
//############################################################################
tonWriteLog(IN:= TRUE, PT := tWriteLog);

IF (tonWriteLog.Q)
THEN
  MessageData.bWriteFile      := TRUE;
  tonWriteLog(IN:= FALSE);
END_IF

//-----------------------------------------------------------------------------------------------------------------
// write message list to file
//-----------------------------------------------------------------------------------------------------------------
MessageData(pList			        := ADR(GVL_MSG.Messages),
			      pLocalTime        := ADR(GVL_MSG.dtLocalTime), 
			      bBusy=> );

// clear write trigger
IF MessageData.bWriteFile AND
   MessageData.bDone
THEN
  MessageData.bWriteFile      := FALSE;
END_IF
//############################################################################
// logging/
//############################################################################



//############################################################################
// Visualization data	
//############################################################################	
// get enumerations from XPU for visu:
eTransportState                       := f_GetState   (GVL_XTS.XtsTransportState.State);
eTransportResult                      := f_GetProgress(GVL_XTS.XtsTransportState.State);

eXpuState                             := f_GetState   (GVL_XTS.XpuState.State);
eXpuResult                            := f_GetProgress(GVL_XTS.XpuState.State);

eXpuCheck                             := GVL_XTS.XpuState.Check;

// display xpu state and result in visu
// get strings and info
sCaGroupState                         := TO_STRING(GVL_XTS.CaGroupInfo.CaGroupState);

sTransportState                       := TO_STRING(eTransportState);
sTransportCheck                       := TO_STRING(GVL_XTS.XtsTransportState.Check);
sTransportResult                      := TO_STRING(eTransportResult);

sXpuState                             := TO_STRING(eXpuState);
sXpuResult                            := TO_STRING(eXpuResult);
sXpuCheck                             := TO_STRING(eXpuCheck);

sXpuOpMode                            := GVL_XTS.Xpu.OpModeToString();
sXpuMoverdetectionMode                := GVL_XTS.Xpu.IdDetectionModeToString();
sXpuMoverAssignement                  := GVL_XTS.Xpu.MoverPositionAssignementToString();

nMoverSelected                        := SEL((nMoverSelected<1), nMoverSelected, 1);
nMoverSelected                        := SEL((nMoverSelected>MAX_MOVER), nMoverSelected, MAX_MOVER);

nStationSelected                      := SEL((nStationSelected<1), nStationSelected, 1);
nStationSelected                      := SEL((nStationSelected>MAX_STATION), nStationSelected, MAX_STATION);

bStationEnable                        := SEL((GVL_XTS.StationCtrl[nStationSelected].eCmd = E_STATION_CTRL.STATION_ENABLE),        FALSE, TRUE);
bStationEnter                         := SEL((GVL_XTS.StationCtrl[nStationSelected].eCmd = E_STATION_CTRL.STATION_MOVER_ENTER),   FALSE, TRUE);
bStationStart                         := SEL((GVL_XTS.StationCtrl[nStationSelected].eCmd = E_STATION_CTRL.STATION_PROCESS_START), FALSE, TRUE);
bStationDone                          := SEL((GVL_XTS.StationCtrl[nStationSelected].eCmd = E_STATION_CTRL.STATION_PROCESS_DONE),  FALSE, TRUE);
bStationOut                           := SEL((GVL_XTS.StationCtrl[nStationSelected].eCmd = E_STATION_CTRL.STATION_MOVER_OUT),     FALSE, TRUE);
bStationGone                          := SEL((GVL_XTS.StationCtrl[nStationSelected].eCmd = E_STATION_CTRL.STATION_MOVER_GONE),    FALSE, TRUE);

eMoverState                           := f_GetState   (GVL_XTS.MoverState[nMoverSelected].State);
eMoverResult                          := f_GetProgress(GVL_XTS.MoverState[nMoverSelected].State);

sMoverState                           := TO_STRING(eMoverState);
sMoverResult                          := TO_STRING(eMoverResult);

sStationState                         := TO_STRING(GVL_XTS.StationState[nStationSelected].eState);
sStationStateMask                     := Tc2_Utilities.BYTE_TO_BINSTR(GVL_XTS.StationState[nStationSelected].nMask, 8);
sStationCtrlMask                      := Tc2_Utilities.BYTE_TO_BINSTR(GVL_XTS.StationCtrl[nStationSelected].nMask, 8);

tStationSelectedQueue                 := GVL_XTS.StationQueue[nStationSelected];

ACTION StationParameterInit:
//-----------------------------------------------------------------------------
//
//  HAUD 2024.04.11
//
//  - hard coded station parameters as example
//  - TODO: xml DataServer implementation for station parameter read/write
//
//  - reminder: (this you HAVE to check manually when setting up the transport)
//-----------------------------------------------------------------------------
//    - DO NOT place the modulo turn within the range of a station
//
//    - in case the extern process requires multiple xts stations, 
//      - the range must be closed and in strict order
//-----------------------------------------------------------------------------
//-----------------------------------------------------------------------------

//-----------------------------------------------------------------------------------------------------------------------------------------
nStationParameter := 1;
GVL_XTS.StationParameter[nStationParameter].rPosWait              :=    140.0; // absolute modulo position

GVL_XTS.StationParameter[nStationParameter].nConfiguredStopCount  :=      1;   // how many stops the mover has to make in this station
GVL_XTS.StationParameter[nStationParameter].rPosStop[1]           :=    235.0; // relative to rPosWait

GVL_XTS.StationParameter[nStationParameter].rReleaseDistance      :=     75.0; // relative to Mover.ActPos

GVL_XTS.StationParameter[nStationParameter].rGap                  :=    105.0;
GVL_XTS.StationParameter[nStationParameter].rVelo                 :=   1250.0;
GVL_XTS.StationParameter[nStationParameter].rAccDec               :=  17500.0;
GVL_XTS.StationParameter[nStationParameter].rJerk                 := 600000.0;

//-----------------------------------------------------------------------------------------------------------------------------------------
nStationParameter := 2;
GVL_XTS.StationParameter[nStationParameter].rPosWait              :=   1890.0; // absolute modulo position

GVL_XTS.StationParameter[nStationParameter].nConfiguredStopCount  :=      1;   // how many stops the mover has to make in this station
GVL_XTS.StationParameter[nStationParameter].rPosStop[1]           :=    235.0; // relative to rPosWait

GVL_XTS.StationParameter[nStationParameter].rReleaseDistance      :=    350.0; // relative to Mover.ActPos

GVL_XTS.StationParameter[nStationParameter].rGap                  :=    105.0;
GVL_XTS.StationParameter[nStationParameter].rVelo                 :=   1250.0;
GVL_XTS.StationParameter[nStationParameter].rAccDec               :=  17500.0;
GVL_XTS.StationParameter[nStationParameter].rJerk                 := 600000.0;

//-----------------------------------------------------------------------------------------------------------------------------------------
nStationParameter := 3;
GVL_XTS.StationParameter[nStationParameter].rPosWait              :=   2640.0; // absolute modulo position

GVL_XTS.StationParameter[nStationParameter].nConfiguredStopCount  :=      1;   // how many stops the mover has to make in this station
GVL_XTS.StationParameter[nStationParameter].rPosStop[1]           :=    235.0; // relative to rPosWait

GVL_XTS.StationParameter[nStationParameter].rReleaseDistance      :=    150.0; // relative to Mover.ActPos

GVL_XTS.StationParameter[nStationParameter].rGap                  :=    105.0;
GVL_XTS.StationParameter[nStationParameter].rVelo                 :=   1500.0;
GVL_XTS.StationParameter[nStationParameter].rAccDec               :=  17500.0;
GVL_XTS.StationParameter[nStationParameter].rJerk                 := 600000.0;

//-----------------------------------------------------------------------------------------------------------------------------------------
nStationParameter := 4;
GVL_XTS.StationParameter[nStationParameter].rPosWait              :=   3640.0; // absolute modulo position

GVL_XTS.StationParameter[nStationParameter].nConfiguredStopCount  :=      1;   // how many stops the mover has to make in this station
GVL_XTS.StationParameter[nStationParameter].rPosStop[1]           :=    235.0; // relative to rPosWait

GVL_XTS.StationParameter[nStationParameter].rReleaseDistance      :=    100.0; // relative to Mover.ActPos

GVL_XTS.StationParameter[nStationParameter].rGap                  :=    105.0;
GVL_XTS.StationParameter[nStationParameter].rVelo                 :=   1500.0;
GVL_XTS.StationParameter[nStationParameter].rAccDec               :=  17500.0;
GVL_XTS.StationParameter[nStationParameter].rJerk                 := 600000.0;

//-----------------------------------------------------------------------------------------------------------------------------------------
nStationParameter := 5;
GVL_XTS.StationParameter[nStationParameter].rPosWait              :=   4890.0; // absolute modulo position

GVL_XTS.StationParameter[nStationParameter].nConfiguredStopCount  :=      1;   // how many stops the mover has to make in this station
GVL_XTS.StationParameter[nStationParameter].rPosStop[1]           :=    235.0; // relative to rPosWait

GVL_XTS.StationParameter[nStationParameter].rReleaseDistance      :=     50.0; // relative to Mover.ActPos

GVL_XTS.StationParameter[nStationParameter].rGap                  :=    105.0;
GVL_XTS.StationParameter[nStationParameter].rVelo                 :=   1500.0;
GVL_XTS.StationParameter[nStationParameter].rAccDec               :=  17500.0;
GVL_XTS.StationParameter[nStationParameter].rJerk                 := 600000.0;
END_ACTION

END_PROGRAM

// ---- MAPPING/MAPPING_out.TcPOU
PROGRAM MAPPING_out
VAR CONSTANT
{IF defined (MOVER_MAP)}
  {info 'MAPPING_out - MOVER_MAPPING active'}
  bBypassMappingMover       : BOOL  := FALSE;
{ELSE}
  bBypassMappingMover       : BOOL  := TRUE;
{END_IF}
{IF defined (STATION_MAP)}
  {info 'MAPPING_out - STATION_MAPPING active'}
  bBypassMappingStation     : BOOL  := FALSE;
{ELSE}
  bBypassMappingStation     : BOOL  := TRUE;
{END_IF}
END_VAR
VAR
  bFirstCycle       : BOOL := TRUE;
{IF defined (MOVER_MAP)}
  MoverState        : U_MOVER_STATE;
  MoverInfo         : U_MOVER_INFO;

{ELSE}
  MoverState        : BYTE;
  MoverInfo         : BYTE;
{END_IF}
{IF defined (STATION_MAP)}
  StationState      : U_XTS_STATION_STATE;
{ELSE}
  StationState      : BYTE;
{END_IF}

  TransportState    : U_XTS_TRANSPORT_STATE;

  szMoverInfo,
  szMoverState        : ARRAY[1..2] OF UDINT;

  szStationState      : ARRAY[1..2] OF UDINT;

  szTransportState    : ARRAY[1..2] OF UDINT;
END_VAR


IF (bFirstCycle)
THEN
  bFirstCycle         := FALSE;
  
  szMoverState[1]     := SIZEOF(MoverState);
  szMoverState[2]     := SIZEOF(GVL_XTS.MoverState);
  
  szMoverInfo [1]     := SIZEOF(MoverInfo);
  szMoverInfo [2]     := SIZEOF(GVL_XTS.MoverInfo);
  
  szStationState [1]  := SIZEOF(StationState);
  szStationState [2]  := SIZEOF(GVL_XTS.StationState);
  
  
  szTransportState [1]:= SIZEOF(TransportState);
  szTransportState [2]:= SIZEOF(GVL_XTS.XtsTransportState);
END_IF

IF NOT bBypassMappingMover
THEN
  memcpy(ADR(MoverState),      ADR(GVL_XTS.MoverState),         SIZEOF(MoverState));
  memcpy(ADR(MoverInfo),       ADR(GVL_XTS.MoverInfo),          SIZEOF(MoverInfo));
END_IF

IF NOT bBypassMappingStation
THEN
  memcpy(ADR(StationState),    ADR(GVL_XTS.StationState),       SIZEOF(StationState));
END_IF

  memcpy(ADR(TransportState),  ADR(GVL_XTS.XtsTransportState),  SIZEOF(TransportState));

END_PROGRAM

// ---- MSG/f_MessageSet.TcPOU
FUNCTION f_MessageSet : BOOL
VAR_INPUT
  stMessage   : ST_Message;
END_VAR
VAR
  _uiIndex   : UINT;
END_VAR

stMessage.tTime                     := GVL_MSG.sLocalTime;

FOR _uiIndex := 1 TO GVL_MSG.MAX_MESSAGE
DO
  IF (GVL_MSG.Messages[_uiIndex].eType = e_MessageType.eMessageEmpty)
  THEN
    GVL_MSG.Messages[_uiIndex]      := stMessage;
    GVL_MSG.MessageIndex             := _uiIndex;
    EXIT;
  END_IF
END_FOR

IF (stMessage.eType = E_MessageType.eMessageError)
THEN
  // in case of error: increment counter
  GVL_MSG.MessageError := GVL_MSG.MessageError + 1;
END_IF

END_FUNCTION

// ---- XTS/CaGroup/FB_CaGroup.TcPOU
//---------------------------------------------------------------------------------------------------------------
//
//  HAUD 2023.12.13
//
//
//  fb_CaGroup
//  - handles CA group states
//  - add mover to group
//  - remove mover from group
//  - clear group error
//  - startup procedure for getting group ready to work
//
//
//  VAR INPUT / OUTPUT --> see properties
//
//---------------------------------------------------------------------------------------------------------------//
// This SOFTWARE is provided as an Exemple by THE PROVIDER "as is" and "with all faults." THE PROVIDER makes no  //
// representations or warranties of any kind concerning the safety, suitability, lack of viruses, inaccuracies,  //
// typographical errors, or other harmful components of this SOFTWARE. There are inherent dangers in the use of  //
// any software, and you are solely responsible for determining whether this SOFTWARE is compatible with your    //
// equipment and other software installed on your equipment. You are also solely responsible for the protection  //
// of your equipment and backup of your data, and THE PROVIDER will not be liable for any damages you may suffer //
// in connection with using, modifying, or distributing this SOFTWARE.                                           //
//---------------------------------------------------------------------------------------------------------------//
FUNCTION_BLOCK FB_CaGroup	IMPLEMENTS I_XtsTransport_CaGroup
VAR CONSTANT
{attribute 'hide'} 
  GROUP_HALT_JERK             : LREAL := 500_000.0;
{attribute 'hide'} 
  GROUP_HALT_DEC              : LREAL :=  12_500.0;
END_VAR
VAR
  _eCheck                     : E_GROUP_CHECK;
  _bError                     : BOOL;

  _GroupRef                   : REFERENCE TO Tc3_McCoordinatedMotion.AXES_GROUP_REF;

  _AxisRefMover               : REFERENCE TO ARRAY[1..MAX_MOVER] OF Tc2_MC2.AXIS_REF;
  _MoverItf                   : REFERENCE TO ARRAY[1..MAX_MOVER] OF I_XtsTransport_Mover;  // mover methods

  _stMoveData                 : ST_MOVE_DATA; // dyn constraints for _MoverItf[i].Halt(Execute, stMoveData)

  // CA group fb instances
  _fbAddAxisGroup             : ARRAY[1..MAX_MOVER] OF Tc3_McCoordinatedMotion.MC_AddAxisToGroup;
  _fbRemoveAxisGroup          : ARRAY[1..MAX_MOVER] OF Tc3_McCoordinatedMotion.MC_RemoveAxisFromGroup;

  _fbGroupDisable             : Tc3_McCoordinatedMotion.MC_GroupDisable;
  _fbGroupEnable              : Tc3_McCoordinatedMotion.MC_GroupEnable;
  _fbGroupErrorRead           : Tc3_McCoordinatedMotion.MC_GroupReadError;
  _fbGroupStatusRead          : Tc3_McCoordinatedMotion.MC_GroupReadStatus;
  _fbGroupReset               : Tc3_McCoordinatedMotion.MC_GroupReset;
  _fbGroupStop                : Tc3_McCoordinatedMotion.MC_GroupStop;

  _stGroupInfo                : ST_GROUP_INFO;  // additional bits about the state of the CA group

  _rtrigGroupStatusRead,
  _rtrigGroupErrorRead        : Tc2_Standard.R_TRIG;

  _stMsg                      : ST_Message;
  _eMessageLevel              : E_MessageType;
END_VAR

METHOD AddAll : E_PROGRESS
VAR_INPUT
  Execute     : BOOL;
END_VAR
VAR_INST
  _nErrorId   : UDINT;
  _eState     : E_PROGRESS;

  _nMover     : UINT;
END_VAR
IF NOT Execute THEN _eState     := E_PROGRESS.PROGRESS_INIT; END_IF 
IF NOT Check() THEN AddAll := E_PROGRESS.PROGRESS_ERROR; RETURN; END_IF


CASE _eState
OF
  E_PROGRESS.PROGRESS_INIT:
    IF Execute
    THEN
      _nErrorId               := 0;
      _nMover                 := 1;

      IF (_stGroupInfo.AxisCount < MAX_MOVER)
      THEN
        _eState               := E_PROGRESS.PROGRESS_BUSY;

      ELSE
        _eState               := E_PROGRESS.PROGRESS_DONE;

        IF (_eMessageLevel = E_MessageType.eMessageVerbose)
        THEN
          _stMsg.eType        := E_MessageType.eMessageVerbose;
          _stMsg.eSubdevice   := e_Subdevice.fbGroupAddAxis;
          _stMsg.iErrorNumber := _nMover;
          _stMsg.sText        := TO_STRING(_eState);
          f_MessageSet(_stMsg);
        END_IF
      END_IF
    END_IF
END_CASE
//-----------------------------------------------------------------------------
//-----------------------------------------------------------------------------
CASE _eState
OF
  E_PROGRESS.PROGRESS_BUSY:
    IF (_eMessageLevel = E_MessageType.eMessageVerbose)
    THEN
      _stMsg.eType            := E_MessageType.eMessageVerbose;
      _stMsg.eSubdevice       := e_Subdevice.fbGroupAddAxis;
      _stMsg.iErrorNumber     := _nMover;
      _stMsg.sText            := TO_STRING(_eState);
      f_MessageSet(_stMsg);
    END_IF

    _eState                   := E_PROGRESS.PROGRESS_PREPARE;
    _fbAddAxisGroup[_nMover](
                AxesGroup     := _GroupRef, 
                Axis          := _AxisRefMover[_nMover], 
                Execute       := FALSE, 
                IdentInGroup  := UDINT_TO_IDENTINGROUP(_AxisRefMover[_nMover].NcToPlc.AxisId));
END_CASE
//-----------------------------------------------------------------------------
//-----------------------------------------------------------------------------
CASE _eState
OF
  E_PROGRESS.PROGRESS_PREPARE:
    _fbAddAxisGroup[_nMover](
                AxesGroup     := _GroupRef, 
                Axis          := _AxisRefMover[_nMover], 
                Execute       := TRUE, 
                IdentInGroup  := UDINT_TO_IDENTINGROUP(_AxisRefMover[_nMover].NcToPlc.AxisId));

    IF (_fbAddAxisGroup[_nMover].Error)
    THEN
      _eState                 := E_PROGRESS.PROGRESS_ERROR;
      _nErrorId               := _fbAddAxisGroup[_nMover].ErrorId;

      _stMsg.eType            := E_MessageType.eMessageError;
      _stMsg.eSubdevice       := e_Subdevice.fbGroupAddAxis;
      _stMsg.iErrorNumber     := _nErrorId;
      _stMsg.sText            := TO_STRING(_eState);
      f_MessageSet(_stMsg);

    ELSIF (_fbAddAxisGroup[_nMover].Done)
    THEN
      _eState                 := E_PROGRESS.PROGRESS_CHECK;

      IF (_eMessageLevel = E_MessageType.eMessageVerbose)
      THEN
        _stMsg.eType          := E_MessageType.eMessageVerbose;
        _stMsg.eSubdevice     := e_Subdevice.fbGroupAddAxis;
        _stMsg.iErrorNumber   := _nMover;
        _stMsg.sText          := TO_STRING(_eState);
        f_MessageSet(_stMsg);
      END_IF
    END_IF
END_CASE
//-----------------------------------------------------------------------------
//-----------------------------------------------------------------------------
CASE _eState
OF
  E_PROGRESS.PROGRESS_CHECK:
    _eState                   := E_PROGRESS.PROGRESS_OCCUPIED;
    _fbAddAxisGroup[_nMover](
                AxesGroup     := _GroupRef, 
                Axis          := _AxisRefMover[_nMover], 
                Execute       := FALSE, 
                IdentInGroup  := UDINT_TO_IDENTINGROUP(_AxisRefMover[_nMover].NcToPlc.AxisId));
END_CASE
//-----------------------------------------------------------------------------
//-----------------------------------------------------------------------------
CASE _eState
OF
  E_PROGRESS.PROGRESS_OCCUPIED:
    IF (_nMover > MAX_MOVER-1)
    THEN
      _eState                 := E_PROGRESS.PROGRESS_DONE;

      IF (_eMessageLevel > E_MessageType.eMessageError)
      THEN
        _stMsg.eType          := E_MessageType.eMessageInfo;
        _stMsg.eSubdevice     := e_Subdevice.fbGroupAddAxis;
        _stMsg.iErrorNumber   := MAX_MOVER;
        _stMsg.sText          := TO_STRING(_eState);
        f_MessageSet(_stMsg);
      END_IF
    ELSE
      _nMover                 := _nMover + 1;
      _eState                 := E_PROGRESS.PROGRESS_BUSY;
    END_IF
END_CASE
//-----------------------------------------------------------------------------
//-----------------------------------------------------------------------------

AddAll                   := _eState;
END_METHOD

PROPERTY AxisRef : REFERENCE TO ARRAY[1..MAX_MOVER] OF Tc2_MC2.AXIS_REF
SET
_AxisRefMover REF= AxisRef;
END_SET
END_PROPERTY

METHOD PROTECTED Check : BOOL

IF NOT __ISVALIDREF(_GroupRef)
THEN
  _eCheck                     := E_GROUP_CHECK.CHECK_GROUP_REF_INVALID;
  RETURN;
END_IF

IF NOT __ISVALIDREF(_AxisRefMover)
THEN
  _eCheck                     := E_GROUP_CHECK.CHECK_AXIS_REF_INVALID;
  RETURN;
END_IF

IF NOT __ISVALIDREF(_MoverItf)
THEN
  _eCheck                     := E_GROUP_CHECK.CHECK_Mover_ITF_REF_INVALID;
  RETURN;
END_IF

_eCheck                       := E_GROUP_CHECK.CHECK_DONE;
Check                         := TRUE;
END_METHOD

METHOD Disable : E_PROGRESS
VAR_INPUT
  Execute     : BOOL;
END_VAR
VAR_INST
  _nErrorId   : UDINT;
  _eState     : E_PROGRESS;

  _nMover     : UINT;
END_VAR
IF NOT Execute THEN _eState       := E_PROGRESS.PROGRESS_INIT; END_IF 
IF NOT Check() THEN Disable  := E_PROGRESS.PROGRESS_ERROR; RETURN; END_IF


CASE _eState
OF
  E_PROGRESS.PROGRESS_INIT:
    IF Execute
    THEN
      _nErrorId               := 0;
      _nMover                 := 1;
      _eState                 := E_PROGRESS.PROGRESS_BUSY;
    END_IF
END_CASE
//-----------------------------------------------------------------------------
//-----------------------------------------------------------------------------
CASE _eState
OF
  E_PROGRESS.PROGRESS_BUSY:
    IF (_stGroupInfo.CaGroupState = E_CA_GROUP_STATE.mcGroupStateDisabled)
    THEN
      _eState                 := E_PROGRESS.PROGRESS_DONE;

      IF (_eMessageLevel = E_MessageType.eMessageVerbose)
      THEN
        _stMsg.eType          := E_MessageType.eMessageVerbose;
        _stMsg.eSubdevice     := e_Subdevice.fbGroupDisable;
        _stMsg.iErrorNumber   := _nErrorId;
        _stMsg.sText          := TO_STRING(_eState);
        f_MessageSet(_stMsg);
      END_IF
    ELSE
      _eState                 := E_PROGRESS.PROGRESS_PREPARE;
      _fbGroupDisable(
                AxesGroup     := _GroupRef, 
                Execute       := FALSE);

      _fbGroupReset(
                AxesGroup     := _GroupRef, 
                Execute       := FALSE);
  
      IF (_eMessageLevel = E_MessageType.eMessageVerbose)
      THEN
        _stMsg.eType          := E_MessageType.eMessageVerbose;
        _stMsg.eSubdevice     := e_Subdevice.fbGroupDisable;
        _stMsg.iErrorNumber   := _nErrorId;
        _stMsg.sText          := TO_STRING(_eState);
        f_MessageSet(_stMsg);
      END_IF
    END_IF
END_CASE
//-----------------------------------------------------------------------------
//-----------------------------------------------------------------------------
CASE _eState
OF
  E_PROGRESS.PROGRESS_PREPARE:
    _fbGroupReset(
                AxesGroup     := _GroupRef, 
                Execute       := TRUE);

    IF (_fbGroupReset.Error)
    THEN
      _eState                 := E_PROGRESS.PROGRESS_ERROR;
      _nErrorId               := _fbGroupReset.ErrorId;

      _stMsg.eType            := E_MessageType.eMessageError;
      _stMsg.eSubdevice       := e_Subdevice.fbGroupReset;
      _stMsg.iErrorNumber     := _nErrorId;
      _stMsg.sText            := TO_STRING(_eState);
      f_MessageSet(_stMsg);

      _fbGroupReset(
                AxesGroup     := _GroupRef, 
                Execute       := FALSE);
    ELSE
      IF (_fbGroupReset.Done)
      THEN
        _eState               := E_PROGRESS.PROGRESS_STARTUP;
        _fbGroupReset(
                AxesGroup     := _GroupRef, 
                Execute       := FALSE);
      END_IF
    END_IF
END_CASE
//-----------------------------------------------------------------------------
//-----------------------------------------------------------------------------
CASE _eState
OF
  E_PROGRESS.PROGRESS_STARTUP:
    _fbGroupDisable(
              AxesGroup       := _GroupRef, 
              Execute         := TRUE); 

    IF (_fbGroupDisable.Error)
    THEN
      _eState                 := E_PROGRESS.PROGRESS_ERROR;
      _nErrorId               := _fbGroupDisable.ErrorId;

      _stMsg.eType            := E_MessageType.eMessageError;
      _stMsg.eSubdevice       := e_Subdevice.fbGroupDisable;
      _stMsg.iErrorNumber     := _nErrorId;
      _stMsg.sText            := TO_STRING(_eState);
      f_MessageSet(_stMsg);

      _fbGroupDisable(
              AxesGroup       := _GroupRef, 
              Execute         := FALSE); 


    ELSIF (_fbGroupDisable.Done)
    THEN
      _eState                 := E_PROGRESS.PROGRESS_DONE;

      IF (_eMessageLevel > E_MessageType.eMessageError)
      THEN
        _stMsg.eType          := E_MessageType.eMessageInfo;
        _stMsg.eSubdevice     := e_Subdevice.fbGroupDisable;
        _stMsg.iErrorNumber   := _nErrorId;
        _stMsg.sText          := TO_STRING(_eState);
        f_MessageSet(_stMsg);
      END_IF

      _fbGroupDisable(
              AxesGroup       := _GroupRef, 
              Execute         := FALSE); 
    END_IF
END_CASE
//-----------------------------------------------------------------------------
//-----------------------------------------------------------------------------

Disable                  := _eState;
END_METHOD

METHOD Enable : E_PROGRESS
VAR_INPUT
  Execute     : BOOL;
END_VAR
VAR_INST
  _nErrorId   : UDINT;
  _eState     : E_PROGRESS;

  _nMover     : UINT;
END_VAR
IF NOT Execute THEN _eState       := E_PROGRESS.PROGRESS_INIT; END_IF 
IF NOT Check() THEN Enable   := E_PROGRESS.PROGRESS_ERROR; RETURN; END_IF


CASE _eState
OF
  E_PROGRESS.PROGRESS_INIT:
    IF Execute
    THEN
      _nErrorId               := 0;
      _nMover                 := 1;
      _eState                 := E_PROGRESS.PROGRESS_BUSY;
    END_IF
END_CASE
//-----------------------------------------------------------------------------
//-----------------------------------------------------------------------------
CASE _eState
OF
  E_PROGRESS.PROGRESS_BUSY:
    _eState                   := E_PROGRESS.PROGRESS_PREPARE;
    _fbGroupEnable(
                AxesGroup     := _GroupRef, 
                Execute       := FALSE);

    IF (_eMessageLevel = E_MessageType.eMessageVerbose)
    THEN
      _stMsg.eType            := E_MessageType.eMessageVerbose;
      _stMsg.eSubdevice       := e_Subdevice.fbGroupEnable;
      _stMsg.iErrorNumber     := _nErrorId;
      _stMsg.sText            := TO_STRING(_eState);
      f_MessageSet(_stMsg);
    END_IF
END_CASE
//-----------------------------------------------------------------------------
//-----------------------------------------------------------------------------
CASE _eState
OF
  E_PROGRESS.PROGRESS_PREPARE:
    _fbGroupEnable(
                AxesGroup     := _GroupRef, 
                Execute       := TRUE);

    IF (_fbGroupEnable.Error)
    THEN
      _eState                 := E_PROGRESS.PROGRESS_ERROR;
      _nErrorId               := _fbGroupEnable.ErrorId;

      _stMsg.eType            := E_MessageType.eMessageError;
      _stMsg.eSubdevice       := e_Subdevice.fbGroupEnable;
      _stMsg.iErrorNumber     := _nErrorId;
      _stMsg.sText            := TO_STRING(_eState);
      f_MessageSet(_stMsg);

      _fbGroupEnable(
                AxesGroup     := _GroupRef, 
                Execute       := FALSE);

    ELSIF (_fbGroupEnable.Done)
    THEN
      _eState                 := E_PROGRESS.PROGRESS_DONE;

      IF (_eMessageLevel > E_MessageType.eMessageError)
      THEN
        _stMsg.eType          := E_MessageType.eMessageInfo;
        _stMsg.eSubdevice     := e_Subdevice.fbGroupEnable;
        _stMsg.iErrorNumber   := _nErrorId;
        _stMsg.sText          := TO_STRING(_eState);
        f_MessageSet(_stMsg);
      END_IF
      _fbGroupEnable(
                AxesGroup     := _GroupRef, 
                Execute       := FALSE);
    END_IF
END_CASE
//-----------------------------------------------------------------------------
//-----------------------------------------------------------------------------

Enable                   := _eState;
END_METHOD

PROPERTY GroupInfo : reference to ST_GROUP_INFO
GET
GroupInfo REF= _stGroupInfo;
END_GET
END_PROPERTY

PROPERTY GroupRef : reference to Tc3_McCoordinatedMotion.AXES_GROUP_REF
GET
GroupRef REF= _GroupRef;
END_GET
SET
_GroupRef REF= GroupRef;
END_SET
END_PROPERTY

METHOD InfoCycle : DWORD
VAR_INPUT
  EnableCycle          : BOOL;
END_VAR
VAR_INST
  _nErrorIdADS,
  _nErrorIdRead   : UDINT;

  _nIdx           : udint;
END_VAR
IF NOT Check() THEN RETURN; END_IF

_stMsg.eDevice                              := e_Device.CaGroup;

//-----------------------------------------------------------------------------------------------
// cyclic CA group
//-----------------------------------------------------------------------------------------------
_fbGroupStatusRead(
              AxesGroup                     := _GroupRef, 
              Enable                        := EnableCycle, 
              Valid                         => _stGroupInfo.GroupStatusValid, 
              Busy                          => _stGroupInfo.GroupStatusBusy, 
              GroupMoving                   => _stGroupInfo.GroupMoving, 
              GroupHoming                   => _stGroupInfo.GroupHoming, 
              GroupErrorStop                => _stGroupInfo.GroupErrorStop, 
              GroupNotReady                 => _stGroupInfo.GroupNotReady, 
              GroupStandby                  => _stGroupInfo.GroupStandby, 
              GroupStopping                 => _stGroupInfo.GroupStopping, 
              GroupDisabled                 => _stGroupInfo.GroupDisabled, 
              AllAxesStanding               => _stGroupInfo.AllAxesStanding, 
              ConstantVelocity              => _stGroupInfo.ConstantVelocity, 
              Accelerating                  => _stGroupInfo.Accelerating, 
              Decelerating                  => _stGroupInfo.Decelerating, 
              InPosition                    => _stGroupInfo.InPosition, 
              Error                         => _stGroupInfo.GroupError, 
              ErrorId                       => );

_fbGroupErrorRead(
              AxesGroup                     := _GroupRef, 
              Enable                        := EnableCycle, 
              ErrorId                       => , 
              GroupErrorId                  => _stGroupInfo.GroupErrorId);


_stGroupInfo.AxisCount                      := _GroupRef.NcToPlc.CA.Common.GroupAxesCount;
_stGroupInfo.CaGroupOID                     := _GroupRef.NcToPlc.CA.Common.GroupOID;
_stGroupInfo.CaGroupState                   := TO_UINT(_GroupRef.NcToPlc.CA.Common.GroupStatus.State);

_stGroupInfo.AxisCountEnabled               := 0;
FOR _nIdx := 1 TO MAX_MOVER
DO
  IF (_AxisRefMover[_nIdx].Status.ControlLoopClosed)
  THEN
    _stGroupInfo.AxisCountEnabled           := _stGroupInfo.AxisCountEnabled + 1;
  END_IF
END_FOR	
			  
// fetch internal fb error
_rtrigGroupErrorRead(CLK                    := _fbGroupErrorRead.Error);
IF _rtrigGroupErrorRead.Q
THEN
  _nErrorIdADS                              := _fbGroupErrorRead.ErrorId;

  _stMsg.eType                              := E_MessageType.eMessageError;
  _stMsg.eSubdevice                         := e_Subdevice.fbGroupErrorRead;
  _stMsg.iErrorNumber                       := _nErrorIdADS;
  _stMsg.sText                              := '';
  f_MessageSet(_stMsg);
END_IF

// Dyn constrainst for McHaltAll(method)
_stMoveData.rJerk                           := GROUP_HALT_JERK;
_stMoveData.rAcc                            := GROUP_HALT_DEC;
END_METHOD

METHOD McHaltAll : E_PROGRESS
VAR_INPUT
  Execute       : BOOL;
END_VAR
VAR_INST
  _nErrorId     : UDINT;
  _eState       : E_PROGRESS;
  _eResult      : E_PROGRESS;

  _nMover       : UINT;

  _nRepeat      : UINT;
END_VAR
IF NOT Execute 
THEN 
	_eState     := E_PROGRESS.PROGRESS_INIT; 
END_IF 
IF NOT Check() 
THEN 
	McHaltAll   := E_PROGRESS.PROGRESS_ERROR; 
	RETURN; 
END_IF


CASE _eState
OF
  E_PROGRESS.PROGRESS_INIT:
    IF Execute
    THEN
      _fbGroupStop(
              AxesGroup       := _GroupRef, 
              Execute         := FALSE, 
              Deceleration    := GROUP_HALT_DEC, 
              Jerk            := GROUP_HALT_JERK);

      _nErrorId               := 0;
      _nMover                 := 1;
      _eState                 := E_PROGRESS.PROGRESS_BUSY;
    END_IF
END_CASE

//-----------------------------------------------------------------------------
//-----------------------------------------------------------------------------
CASE _eState
OF
  E_PROGRESS.PROGRESS_BUSY:
    IF NOT (_stGroupInfo.CaGroupState = E_CA_GROUP_STATE.mcGroupStateMoving)
    THEN
      _eState                   := E_PROGRESS.PROGRESS_PREPARE;
    ELSE
      _fbGroupStop(
                AxesGroup       := _GroupRef, 
                Execute         := TRUE, 
                Deceleration    := GROUP_HALT_DEC, 
                Jerk            := GROUP_HALT_JERK);
  
      IF (_fbGroupStop.Error)
      THEN
        _stMsg.eType            := E_MessageType.eMessageError;
        _stMsg.eSubdevice       := e_Subdevice.fbGroupStop;
        _stMsg.iErrorNumber     := _fbGroupStop.ErrorId;
        _stMsg.sText            := TO_STRING(_eState);
        f_MessageSet(_stMsg);
  
        _nRepeat                := _nRepeat + 1;
        _eState                 := E_PROGRESS.PROGRESS_PREPARE;
      ELSE
        IF (_fbGroupStop.Done)
        THEN
          IF (_eMessageLevel = E_MessageType.eMessageVerbose)
          THEN
            _stMsg.eType        := E_MessageType.eMessageVerbose;
            _stMsg.eSubdevice   := e_Subdevice.fbGroupStop;
            _stMsg.iErrorNumber := MAX_MOVER;
            _stMsg.sText        := TO_STRING(_eState);
            f_MessageSet(_stMsg);
          END_IF
          _nRepeat              := 0;
          _eState               := E_PROGRESS.PROGRESS_PREPARE;
        END_IF
      END_IF
    END_IF
END_CASE

//-----------------------------------------------------------------------------
//-----------------------------------------------------------------------------
CASE _eState
OF
  E_PROGRESS.PROGRESS_PREPARE:
    _eState                   := E_PROGRESS.PROGRESS_WORKING;
    _fbGroupStop(
              AxesGroup       := _GroupRef, 
              Execute         := FALSE, 
              Deceleration    := GROUP_HALT_DEC, 
              Jerk            := GROUP_HALT_JERK);

    _eResult                  := _MoverItf[_nMover].Reset(FALSE);
    _eResult                  := _MoverItf[_nMover].Halt(FALSE, _stMoveData);
END_CASE
//-----------------------------------------------------------------------------
//-----------------------------------------------------------------------------
CASE _eState
OF
  E_PROGRESS.PROGRESS_WORKING:
    _eResult                  := _MoverItf[_nMover].Halt(TRUE, _stMoveData);

    IF (_eResult = E_PROGRESS.PROGRESS_DONE)
    THEN
      _eResult                := _MoverItf[_nMover].Halt(FALSE, _stMoveData);
      _eState                 := E_PROGRESS.PROGRESS_STARTUP;

    ELSIF (_eResult = E_PROGRESS.PROGRESS_ERROR)
    THEN
      _nErrorId               := _AxisRefMover[_nMover].NcToPlc.ErrorCode;
      _MoverItf[_nMover].Reset(TRUE);

      _stMsg.eType            := E_MessageType.eMessageError;
      _stMsg.eSubdevice       := e_Subdevice.fbHalt;
      _stMsg.iErrorNumber     := _nErrorId;
      _stMsg.sText            := concat( 'McHaltAll: ', TO_STRING(_eResult));
      _stMsg.sText            := concat(_stMsg.sText, ' MoverId: ');
      _stMsg.sText            := concat(_stMsg.sText, TO_STRING(_nMover));
      f_MessageSet(_stMsg);

      _eState                 := E_PROGRESS.PROGRESS_PREPARE;
    END_IF
END_CASE

//-----------------------------------------------------------------------------
//-----------------------------------------------------------------------------
CASE _eState
OF
  E_PROGRESS.PROGRESS_STARTUP:
    IF (_nMover > MAX_MOVER-1)
    THEN
      _eState                 := E_PROGRESS.PROGRESS_CHECK;
    ELSE
      _nMover                 := _nMover + 1;
      _eState                 := E_PROGRESS.PROGRESS_PREPARE;
    END_IF
END_CASE

//-----------------------------------------------------------------------------
//-----------------------------------------------------------------------------
CASE _eState
OF
  E_PROGRESS.PROGRESS_CHECK:
    _eState                   := E_PROGRESS.PROGRESS_DONE;

    IF (_eMessageLevel > E_MessageType.eMessageError)
    THEN
      _stMsg.eType            := E_MessageType.eMessageInfo;
      _stMsg.eSubdevice       := e_Subdevice.fbCaGroup;
      _stMsg.iErrorNumber     := MAX_MOVER;
      _stMsg.sText            := concat('McHaltAll: ', TO_STRING(_eState));
      f_MessageSet(_stMsg);
    END_IF
END_CASE
//-----------------------------------------------------------------------------
//-----------------------------------------------------------------------------
McHaltAll                     := _eState;
END_METHOD

METHOD McResetAll : E_PROGRESS
VAR_INPUT
  Execute       : BOOL;
END_VAR
VAR_INST
  _nErrorId     : UDINT;
  _eRslt,
  _eState       : E_PROGRESS;

  _nMover       : UINT;
END_VAR
IF NOT Execute THEN _eState     := E_PROGRESS.PROGRESS_INIT; END_IF 
IF NOT Check() THEN McResetAll  := E_PROGRESS.PROGRESS_ERROR; RETURN; END_IF


//-----------------------------------------------------------------------------
//-----------------------------------------------------------------------------
CASE _eState
OF
  E_PROGRESS.PROGRESS_INIT:
    IF Execute
    THEN
      _nErrorId                 := 0;
      _nMover                   := 1;

      _eState                   := E_PROGRESS.PROGRESS_BUSY;
    END_IF
END_CASE
//-----------------------------------------------------------------------------
//-----------------------------------------------------------------------------
CASE _eState
OF
  E_PROGRESS.PROGRESS_BUSY:
    _eState                     := E_PROGRESS.PROGRESS_PREPARE;
    _eRslt                      := _MoverItf[_nMover].Reset(FALSE);
END_CASE
//-----------------------------------------------------------------------------
//-----------------------------------------------------------------------------
CASE _eState
OF
  E_PROGRESS.PROGRESS_PREPARE:
    _eRslt                      := _MoverItf[_nMover].Reset(TRUE);

    IF (_eRslt = E_PROGRESS.PROGRESS_ERROR)
    THEN
      _eState                   := E_PROGRESS.PROGRESS_BUSY;

    ELSIF (_eRslt = E_PROGRESS.PROGRESS_DONE)
    THEN
      _eState                   := E_PROGRESS.PROGRESS_STARTUP;
    END_IF
END_CASE
//-----------------------------------------------------------------------------
//-----------------------------------------------------------------------------
CASE _eState
OF
  E_PROGRESS.PROGRESS_STARTUP:
    _eState                     := E_PROGRESS.PROGRESS_CHECK;
    _eRslt                      := _MoverItf[_nMover].Reset(FALSE);
END_CASE
//-----------------------------------------------------------------------------
//-----------------------------------------------------------------------------
CASE _eState
OF
  E_PROGRESS.PROGRESS_CHECK:
    IF (_nMover > MAX_MOVER-1)
    THEN
      _eState                   := E_PROGRESS.PROGRESS_DONE;

      IF (_eMessageLevel = E_MessageType.eMessageVerbose)
      THEN
        _stMsg.eType            := E_MessageType.eMessageVerbose;
        _stMsg.eSubdevice       := e_Subdevice.fbReset;
        _stMsg.iErrorNumber     := 0;
        _stMsg.sText            := concat( 'State: ', TO_STRING(_eState));
        f_MessageSet(_stMsg);
      END_IF
    ELSE
      _nMover                   := _nMover + 1;
      _eState                   := E_PROGRESS.PROGRESS_BUSY;
    END_IF
END_CASE
//-----------------------------------------------------------------------------
//-----------------------------------------------------------------------------


McResetAll                      := _eState;
END_METHOD

PROPERTY MessageLevel : e_messagetype
SET
_eMessageLevel := MessageLevel;
END_SET
END_PROPERTY

PROPERTY MoverItf : reference TO ARRAY[1..MAX_MOVER] OF I_XtsTransport_Mover
SET
_MoverItf REF= MoverItf;
END_SET
END_PROPERTY

METHOD RemoveAll : E_PROGRESS
VAR_INPUT
  Execute     : BOOL;
END_VAR
VAR_INST
  _nErrorId   : UDINT;
  _eState     : E_PROGRESS;

  _nMover     : UINT;
END_VAR
IF NOT Execute THEN _eState         := E_PROGRESS.PROGRESS_INIT; END_IF 
IF NOT Check() THEN RemoveAll  := E_PROGRESS.PROGRESS_ERROR; RETURN; END_IF


CASE _eState
OF
  E_PROGRESS.PROGRESS_INIT:
    IF Execute
    THEN
      _nErrorId               := 0;
      _nMover                 := 1;

      IF (_stGroupInfo.AxisCount > 0)
      THEN
        _eState               := E_PROGRESS.PROGRESS_BUSY;
      ELSE
        _eState               := E_PROGRESS.PROGRESS_DONE;

        IF (_eMessageLevel = E_MessageType.eMessageVerbose)
        THEN
          _stMsg.eType        := E_MessageType.eMessageVerbose;
          _stMsg.eSubdevice   := e_Subdevice.fbGroupRemoveAxis;
          _stMsg.iErrorNumber := _stGroupInfo.AxisCount;
          _stMsg.sText        := TO_STRING(_eState);
          f_MessageSet(_stMsg);
        END_IF
      END_IF
    END_IF
END_CASE
//-----------------------------------------------------------------------------
//-----------------------------------------------------------------------------
CASE _eState
OF
  E_PROGRESS.PROGRESS_BUSY:
    IF (_eMessageLevel = E_MessageType.eMessageVerbose)
    THEN
      _stMsg.eType          := E_MessageType.eMessageVerbose;
      _stMsg.eSubdevice     := e_Subdevice.fbGroupRemoveAxis;
      _stMsg.iErrorNumber   := _nMover;
      _stMsg.sText          := TO_STRING(_eState);
      //f_MessageSet(_stMsg);
    END_IF

    _eState                 := E_PROGRESS.PROGRESS_PREPARE;
    _fbRemoveAxisGroup[_nMover](
            AxesGroup       := _GroupRef, 
            Execute         := FALSE,
            IdentInGroup    := UDINT_TO_IDENTINGROUP(_AxisRefMover[_nMover].NcToPlc.AxisId));
END_CASE
//-----------------------------------------------------------------------------
//-----------------------------------------------------------------------------
CASE _eState
OF
  E_PROGRESS.PROGRESS_PREPARE:
    _fbRemoveAxisGroup[_nMover](
              AxesGroup       := _GroupRef, 
              Execute         := TRUE,
              IdentInGroup    := UDINT_TO_IDENTINGROUP(_AxisRefMover[_nMover].NcToPlc.AxisId));

    IF (_fbRemoveAxisGroup[_nMover].Error)
    THEN
      _eState                 := E_PROGRESS.PROGRESS_ERROR;
      _nErrorId               := _fbRemoveAxisGroup[_nMover].ErrorId;

      _stMsg.eType            := E_MessageType.eMessageError;
      _stMsg.eSubdevice       := e_Subdevice.fbGroupRemoveAxis;
      _stMsg.iErrorNumber     := _nErrorId;
      _stMsg.sText            := TO_STRING(_eState);
      f_MessageSet(_stMsg);

    ELSIF (_fbRemoveAxisGroup[_nMover].Done)
    THEN
      _eState                 := E_PROGRESS.PROGRESS_CHECK;

      IF (_eMessageLevel = E_MessageType.eMessageVerbose)
      THEN
        _stMsg.eType          := E_MessageType.eMessageVerbose;
        _stMsg.eSubdevice     := e_Subdevice.fbGroupRemoveAxis;
        _stMsg.iErrorNumber   := _nMover;
        _stMsg.sText          := TO_STRING('DONE');
        //f_MessageSet(_stMsg);
      END_IF
    END_IF
END_CASE
//-----------------------------------------------------------------------------
//-----------------------------------------------------------------------------
CASE _eState
OF
  E_PROGRESS.PROGRESS_CHECK:
    _eState                   := E_PROGRESS.PROGRESS_OCCUPIED;
    _fbRemoveAxisGroup[_nMover](
              AxesGroup       := _GroupRef, 
              Execute         := FALSE,
              IdentInGroup    := UDINT_TO_IDENTINGROUP(_AxisRefMover[_nMover].NcToPlc.AxisId));
END_CASE
//-----------------------------------------------------------------------------
//-----------------------------------------------------------------------------
CASE _eState
OF
  E_PROGRESS.PROGRESS_OCCUPIED:
    IF (_nMover > MAX_MOVER-1)
    THEN
      _eState                 := E_PROGRESS.PROGRESS_DONE;

      IF (_eMessageLevel > E_MessageType.eMessageError)
      THEN
        _stMsg.eType          := E_MessageType.eMessageInfo;
        _stMsg.eSubdevice     := e_Subdevice.fbGroupRemoveAxis;
        _stMsg.iErrorNumber   := MAX_MOVER;
        _stMsg.sText          := TO_STRING(_eState);
        f_MessageSet(_stMsg);
      END_IF
    ELSE
      _nMover                 := _nMover + 1;
      _eState                 := E_PROGRESS.PROGRESS_BUSY;
    END_IF
END_CASE
//-----------------------------------------------------------------------------
//-----------------------------------------------------------------------------

RemoveAll                := _eState;
END_METHOD

METHOD Reset : E_PROGRESS
VAR_INPUT
  Execute     : BOOL;
END_VAR
VAR_INST
  _nErrorId   : UDINT;
  _eState     : E_PROGRESS;

  _nMover     : UINT;
END_VAR
IF NOT Execute 
THEN 
	_eState := E_PROGRESS.PROGRESS_INIT; 
END_IF 
IF NOT Check() 
THEN 
	Reset := E_PROGRESS.PROGRESS_ERROR; 
	RETURN; 
END_IF


CASE _eState
OF
  E_PROGRESS.PROGRESS_INIT:
    IF Execute
    THEN
      _nErrorId                 := 0;
      _nMover                   := 1;
      _stGroupInfo.GroupErrorId := 0;
      _stGroupInfo.GroupError   := FALSE;

      _eState                   := E_PROGRESS.PROGRESS_BUSY;
    END_IF
END_CASE
//-----------------------------------------------------------------------------
//-----------------------------------------------------------------------------
CASE _eState
OF
  E_PROGRESS.PROGRESS_BUSY:
    _eState                     := E_PROGRESS.PROGRESS_PREPARE;
    _fbGroupReset(
              AxesGroup         := _GroupRef, 
              Execute           := FALSE);

    IF (_eMessageLevel = E_MessageType.eMessageVerbose)
    THEN
      _stMsg.eType              := E_MessageType.eMessageVerbose;
      _stMsg.eSubdevice         := e_Subdevice.fbGroupReset;
      _stMsg.iErrorNumber       := 0;
      _stMsg.sText              := TO_STRING(_eState);
      //f_MessageSet(_stMsg);
    END_IF
END_CASE
//-----------------------------------------------------------------------------
//-----------------------------------------------------------------------------
CASE _eState
OF
  E_PROGRESS.PROGRESS_PREPARE:
    _fbGroupReset(
              AxesGroup         := _GroupRef, 
              Execute           := TRUE);

    IF (_fbGroupReset.Error)
    THEN
      _eState                   := E_PROGRESS.PROGRESS_ERROR;
      _nErrorId                 := _fbGroupReset.ErrorId;

      _stMsg.eType              := E_MessageType.eMessageError;
      _stMsg.eSubdevice         := e_Subdevice.fbGroupReset;
      _stMsg.iErrorNumber       := _nErrorId;
      _stMsg.sText              := TO_STRING(_eState);
      f_MessageSet(_stMsg);

      _fbGroupReset(
              AxesGroup         := _GroupRef, 
              Execute           := FALSE); 

    ELSIF (_fbGroupReset.Done)
    THEN
      _eState                   := E_PROGRESS.PROGRESS_DONE;

      IF (_eMessageLevel > E_MessageType.eMessageError)
      THEN
        _stMsg.eType            := E_MessageType.eMessageInfo;
        _stMsg.eSubdevice       := e_Subdevice.fbGroupReset;
        _stMsg.iErrorNumber     := _nErrorId;
        _stMsg.sText            := TO_STRING(_eState);
        f_MessageSet(_stMsg);
      END_IF

      _fbGroupReset(
              AxesGroup         := _GroupRef, 
              Execute           := FALSE); 
    END_IF
END_CASE
//-----------------------------------------------------------------------------
//-----------------------------------------------------------------------------

Reset                           := _eState;
END_METHOD

METHOD Stop : E_PROGRESS
VAR_INPUT
  Execute     : BOOL;
END_VAR
VAR_INST
  _nErrorId   : UDINT;
  _eState     : E_PROGRESS;

  _nMover     : UINT;
  _nRepeat    : uint;
END_VAR
IF NOT Execute 
THEN 
	_eState := E_PROGRESS.PROGRESS_INIT; 
END_IF 
IF NOT Check() 
THEN 
	Stop := E_PROGRESS.PROGRESS_ERROR; 
	RETURN; 
END_IF


CASE _eState
OF
  E_PROGRESS.PROGRESS_INIT:
    IF Execute
    THEN
      _nRepeat                  := 0;
      _nErrorId                 := 0;
      _nMover                   := 1;
      _eState                   := E_PROGRESS.PROGRESS_BUSY;
    END_IF
END_CASE
//-----------------------------------------------------------------------------
//-----------------------------------------------------------------------------
CASE _eState
OF
  E_PROGRESS.PROGRESS_BUSY:
    _eState                     := E_PROGRESS.PROGRESS_PREPARE;
    _fbGroupStop(
                AxesGroup       := _GroupRef, 
                Execute         := FALSE, 
                Deceleration    := GROUP_HALT_DEC, 
                Jerk            := GROUP_HALT_JERK);

    IF (_eMessageLevel = E_MessageType.eMessageVerbose)
    THEN
      _stMsg.eType              := E_MessageType.eMessageVerbose;
      _stMsg.eSubdevice         := e_Subdevice.fbGroupStop;
      _stMsg.iErrorNumber       := 0;
      _stMsg.sText              := TO_STRING(_eState);
      f_MessageSet(_stMsg);
    END_IF
END_CASE
//-----------------------------------------------------------------------------
//-----------------------------------------------------------------------------
CASE _eState
OF
  E_PROGRESS.PROGRESS_PREPARE:
    _fbGroupStop(
                AxesGroup       := _GroupRef, 
                Execute         := TRUE, 
                Deceleration    := GROUP_HALT_DEC, 
                Jerk            := GROUP_HALT_JERK);

    IF (_fbGroupStop.Error)
    THEN
      _eState                   := E_PROGRESS.PROGRESS_STARTUP;
      _nErrorId                 := _fbGroupStop.ErrorId;

      _stMsg.eType              := E_MessageType.eMessageError;
      _stMsg.eSubdevice         := e_Subdevice.fbGroupStop;
      _stMsg.iErrorNumber       := _nErrorId;
      _stMsg.sText              := TO_STRING(_eState);
      f_MessageSet(_stMsg);

      _fbGroupReset(
              AxesGroup         := _GroupRef, 
              Execute           := FALSE); 

    ELSIF (_fbGroupStop.Done)
    THEN
      _eState                   := E_PROGRESS.PROGRESS_DONE;

      IF (_eMessageLevel > E_MessageType.eMessageError)
      THEN
        _stMsg.eType            := E_MessageType.eMessageInfo;
        _stMsg.eSubdevice       := e_Subdevice.fbGroupStop;
        _stMsg.iErrorNumber     := _nErrorId;
        _stMsg.sText            := TO_STRING(_eState);
        f_MessageSet(_stMsg);
      END_IF

      _fbGroupStop(
                AxesGroup       := _GroupRef, 
                Execute         := FALSE, 
                Deceleration    := GROUP_HALT_DEC, 
                Jerk            := GROUP_HALT_JERK);
    END_IF
END_CASE
//-----------------------------------------------------------------------------
//-----------------------------------------------------------------------------
CASE _eState
OF
  E_PROGRESS.PROGRESS_STARTUP:
    _fbGroupReset(
              AxesGroup         := _GroupRef, 
              Execute           := TRUE);

    IF (_fbGroupReset.Error)
    THEN
      _nRepeat                  := _nRepeat + 1;
      IF (_nRepeat > 2)
      THEN
        _eState                 := E_PROGRESS.PROGRESS_ERROR;
      END_IF
      _nErrorId                 := _fbGroupReset.ErrorId;

      _stMsg.eType              := E_MessageType.eMessageError;
      _stMsg.eSubdevice         := e_Subdevice.fbGroupStop;
      _stMsg.iErrorNumber       := _nErrorId;
      _stMsg.sText              := TO_STRING(_eState);
      f_MessageSet(_stMsg);

      _fbGroupReset(
              AxesGroup         := _GroupRef, 
              Execute           := FALSE); 

    ELSIF (_fbGroupReset.Done) or not (_fbGroupReset.Busy)
    THEN
      _eState                   := E_PROGRESS.PROGRESS_DONE;

      IF (_eMessageLevel > E_MessageType.eMessageError)
      THEN
        _stMsg.eType            := E_MessageType.eMessageInfo;
        _stMsg.eSubdevice       := e_Subdevice.fbGroupStop;
        _stMsg.iErrorNumber     := _nErrorId;
        _stMsg.sText            := TO_STRING(_eState);
        f_MessageSet(_stMsg);
      END_IF

      _fbGroupReset(
              AxesGroup         := _GroupRef, 
              Execute           := FALSE); 
    END_IF
END_CASE
//-----------------------------------------------------------------------------
//-----------------------------------------------------------------------------

Stop                            := _eState;
END_METHOD

END_FUNCTION_BLOCK

// ---- XTS/Mover/fb_Mover.TcPOU
//---------------------------------------------------------------------------------------------------------------
//
//  HAUD 2023.12.19
//
//  - XTS_TRANSPORT_LAYER
//
//  fb_Mover
//  - all positioning input is modulo value
//  - wrap MC function blocks
//
//
//---------------------------------------------------------------------------------------------------------------
// This SOFTWARE is provided as an Exemple by THE PROVIDER "as is" and "with all faults." THE PROVIDER makes no 
// representations or warranties of any kind concerning the safety, suitability, lack of viruses, inaccuracies, 
// typographical errors, or other harmful components of this SOFTWARE. There are inherent dangers in the use of 
// any software, and you are solely responsible for determining whether this SOFTWARE is compatible with your 
// equipment and other software installed on your equipment. You are also solely responsible for the protection 
// of your equipment and backup of your data, and THE PROVIDER will not be liable for any damages you may suffer 
// in connection with using, modifying, or distributing this SOFTWARE.
//---------------------------------------------------------------------------------------------------------------
FUNCTION_BLOCK fb_Mover IMPLEMENTS I_XtsTransport_Mover
VAR
  _nMoverId         : UINT;

  _sState           : STRING;

  _Master,
  _Mover            : REFERENCE TO AXIS_REF;
  _rLastPosition    : REFERENCE TO LREAL;
  _rLastGap         : REFERENCE TO LREAL;

  _RailLength       : LREAL;
  _nSyncStrategy    : Tc3_Mc3Definitions.MC_SYNC_STRATEGY := Tc3_Mc3Definitions.MC_SYNC_STRATEGY.mcSyncStrategySlow; // minimal movement with this strategy 

  // mover compact axis information
  _stInfo           : REFERENCE TO ST_MOVER_INFO; // ActPos, Enable, ...

  _bError           : BOOL;   // used in Cycle()
  _nErrorIdMover,             // used in Cycle()
  _nErrorIdPower    : UDINT;  // used in Cycle()

  //---------------------------------------------------------------------------
  // MC2 and CA function blocks
  //---------------------------------------------------------------------------
  _wMoverState      : DWORD;

  _fbMoveAbsCa      : Tc3_McCollisionAvoidance.MC_MoveAbsoluteCA;
  _fbGearInPosCa    : Tc3_McCollisionAvoidance.MC_GearInPosCA;
  _fbHaltCa         : Tc3_McCollisionAvoidance.MC_HaltCA;

  _fbMoveAbs        : Tc2_MC2.MC_MoveAbsolute;
  _fbHalt           : Tc2_MC2.MC_Halt;
  _fbReset          : Tc2_MC2.MC_Reset;
  _fbStop           : Tc2_MC2.MC_Stop;

  _fbGearIn         : Tc2_MC2.MC_GearIn;
  _fbGearOut        : Tc2_MC2.MC_GearOut;

  _fbPower          : Tc2_MC2.MC_Power;

  _stMsg            : ST_Message;
  _eMessageLevel    : E_MessageType;
END_VAR

METHOD Check : BOOL
// check The thing that should not be

IF NOT (_nMoverId > 0)
THEN
  _sState                     := 'Mover: missing ID';
  RETURN;
END_IF

IF NOT __ISVALIDREF(_Mover)
THEN
  _sState                     := 'Mover: missing pointer';
  RETURN;
END_IF

IF NOT __ISVALIDREF(_rLastPosition)
THEN
  _sState                     := '_rLastPosition: missing pointer';
  RETURN;
END_IF

IF NOT __ISVALIDREF(_rLastGap)
THEN
  _sState                     := '_rLastGap: missing pointer';
  RETURN;
END_IF

IF NOT __ISVALIDREF(_stInfo)
THEN
  _sState                     := '_stInfo: missing pointer';
  RETURN;
END_IF

_sState                       := 'CHECK_DONE';
Check                         := TRUE;
END_METHOD

METHOD Cycle : E_PROGRESS
VAR_INST
  _eState             : E_PROGRESS;

  _rtrigMoverError,
  _rtrigPowerError    : Tc2_Standard.R_TRIG;
END_VAR
IF NOT Check() THEN Cycle := E_PROGRESS.PROGRESS_ERROR; RETURN; END_IF

_stMsg.eDevice            := e_Device.Mover + _nMoverId;

//-----------------------------------------------------------------------------------------------
// cyclic NC mapping
//-----------------------------------------------------------------------------------------------
_Mover();
//-----------------------------------------------------------------------------------------------


//-----------------------------------------------------------------------------------------------
// cyclic MC_Power
//-----------------------------------------------------------------------------------------------
_fbPower(
        Axis              := _Mover, 
        Enable_Positive   := TRUE, 
        Enable_Negative   := TRUE, 
        BufferMode        := MC_BufferMode.MC_Aborting);

_rtrigPowerError(CLK := _fbPower.Error);
_rtrigMoverError(CLK := _Mover.Status.Error); 

IF _rtrigMoverError.Q
THEN
  _bError                 := TRUE;  // deleted by Reset()
  // catch error
  _nErrorIdMover          := _Mover.Status.ErrorID;
  _stInfo.nErrorId        := _nErrorIdMover;

  _stMsg.eType            := E_MessageType.eMessageError;
  _stMsg.eSubdevice       := e_Subdevice.AxisControl;
  _stMsg.iErrorNumber     := _nErrorIdMover;
  _stMsg.sText            := 'Axis Error';
  f_MessageSet(_stMsg);
END_IF

IF _rtrigPowerError.Q
THEN
  _bError                 := TRUE;  // deleted by Reset()
  // catch error
  _nErrorIdPower          := _fbPower.ErrorID;
  _stInfo.nErrorId        := _nErrorIdPower;

  _stMsg.eType            := E_MessageType.eMessageError;
  _stMsg.eSubdevice       := e_Subdevice.AxisControl;
  _stMsg.iErrorNumber     := _nErrorIdMover;
  _stMsg.sText            := 'Axis Error';
  f_MessageSet(_stMsg);
END_IF
//-----------------------------------------------------------------------------------------------

//-----------------------------------------------------------------------------------------------
// cyclic state
//-----------------------------------------------------------------------------------------------
IF NOT _Mover.Status.ControlLoopClosed
THEN
  _eState                       := E_PROGRESS.PROGRESS_INIT;
ELSE
  _eState                       := E_PROGRESS.PROGRESS_WORKING;
END_IF
 
IF _bError
THEN
  _eState                       := E_PROGRESS.PROGRESS_ERROR;
END_IF
//-----------------------------------------------------------------------------------------------


//-----------------------------------------------------------------------------
// cyclic Mover info data
// get collision avoiding information from cyclic interface
//-----------------------------------------------------------------------------------------------
memcpy(ADR(_wMoverState), ADR(_Mover.NcToPlc.StateDWord2), SIZEOF(_wMoverState));

_stInfo.bMoverEnabled           := _Mover.Status.ControlLoopClosed;
_stInfo.bMoverError             := _bError;
_stInfo.bMoverCoupled           := _Mover.Status.Coupled;
_stInfo.bMoverStandstill        := _Mover.Status.NotMoving;
_stInfo.bMoverAvoidingCollision := _wMoverState.0;

_stInfo.rModuloActPos           := TO_REAL(_Mover.NcToPlc.ModuloActPos);
_stInfo.rAbsActPos              := TO_REAL(_Mover.NcToPlc.ActPos);

_stInfo.rModuloTargetPos        := TO_REAL(Tc2_Math.LMOD(_rLastPosition, _RailLength));
_stInfo.rAbsTargetPos           := TO_REAL(_rLastPosition);

IF (_Mover.NcToPlc.ActPos < _rLastPosition + 0.05) AND
   (_Mover.NcToPlc.ActPos > _rLastPosition - 0.05)
THEN
  _stInfo.bMoverInTarget        := TRUE;
ELSE
  _stInfo.bMoverInTarget        := FALSE;
END_IF
//-----------------------------------------------------------------------------

Cycle                           := _eState;
END_METHOD

METHOD Disable : E_PROGRESS
VAR_INPUT
  Execute             : BOOL;
END_VAR
VAR_INST
  _nErrorId           : UDINT;
  _eState             : E_PROGRESS;
END_VAR
IF NOT Execute THEN _eState  := E_PROGRESS.PROGRESS_INIT; END_IF 
IF NOT Check() THEN Disable  := E_PROGRESS.PROGRESS_ERROR; RETURN; END_IF


CASE _eState
OF
  E_PROGRESS.PROGRESS_INIT:
    IF Execute
    THEN
      _nErrorId               := 0;
      _eState                 := E_PROGRESS.PROGRESS_BUSY;
    END_IF
END_CASE
//-----------------------------------------------------------------------------
//-----------------------------------------------------------------------------
CASE _eState
OF
  E_PROGRESS.PROGRESS_BUSY:
    _eState                   := E_PROGRESS.PROGRESS_PREPARE;
    _fbPower.Enable           := FALSE;
END_CASE
//-----------------------------------------------------------------------------
//-----------------------------------------------------------------------------
CASE _eState
OF
  E_PROGRESS.PROGRESS_PREPARE:
    IF (_fbPower.Error)
    THEN
      _eState                 := E_PROGRESS.PROGRESS_ERROR;
      _nErrorId               := _fbPower.ErrorId;

      _stMsg.eType            := E_MessageType.eMessageError;
      _stMsg.eSubdevice       := e_Subdevice.fbPower;
      _stMsg.iErrorNumber     := _nErrorId;
      _stMsg.sText            := concat('Axis Disable: ', TO_STRING(_eState));
      f_MessageSet(_stMsg);

    ELSIF NOT (_Mover.Status.ControlLoopClosed)
    THEN
      _eState                 := E_PROGRESS.PROGRESS_DONE;

      IF (_eMessageLevel > E_MessageType.eMessageWarning)
      THEN
        _stMsg.eType          := E_MessageType.eMessageVerbose;
        _stMsg.eSubdevice     := e_Subdevice.fbPower;
        _stMsg.iErrorNumber   := 0;
        _stMsg.sText          := concat('Axis Disable: ', TO_STRING(_eState));
        f_MessageSet(_stMsg);
      END_IF
    END_IF
END_CASE
//-----------------------------------------------------------------------------
//-----------------------------------------------------------------------------

Disable                       := _eState;
END_METHOD

METHOD Enable : E_PROGRESS
VAR_INPUT
  Execute             : BOOL;
END_VAR
VAR_INST
  _nErrorId           : UDINT;
  _eState             : E_PROGRESS;
END_VAR
IF NOT Execute THEN _eState  := E_PROGRESS.PROGRESS_INIT; END_IF 
IF NOT Check() THEN Enable   := E_PROGRESS.PROGRESS_ERROR; RETURN; END_IF


CASE _eState
OF
  E_PROGRESS.PROGRESS_INIT:
    IF Execute
    THEN
      _nErrorId               := 0;
      _eState                 := E_PROGRESS.PROGRESS_BUSY;
    END_IF
END_CASE
//-----------------------------------------------------------------------------
//-----------------------------------------------------------------------------
CASE _eState
OF
  E_PROGRESS.PROGRESS_BUSY:
    _eState                   := E_PROGRESS.PROGRESS_PREPARE;
    _fbPower.Enable           := TRUE;
END_CASE
//-----------------------------------------------------------------------------
//-----------------------------------------------------------------------------
CASE _eState
OF
  E_PROGRESS.PROGRESS_PREPARE:
    IF (_fbPower.Error)
    THEN
      _eState                 := E_PROGRESS.PROGRESS_ERROR;
      _nErrorId               := _fbPower.ErrorId;
      _stInfo.nErrorId        := _nErrorId;

      _stMsg.eType            := E_MessageType.eMessageError;
      _stMsg.eSubdevice       := e_Subdevice.fbPower;
      _stMsg.iErrorNumber     := _nErrorId;
      _stMsg.sText            := concat('Axis Enable: ', TO_STRING(_eState));
      f_MessageSet(_stMsg);

    ELSIF (_Mover.Status.ControlLoopClosed)
    THEN
      _eState                 := E_PROGRESS.PROGRESS_DONE;

      IF (_eMessageLevel = E_MessageType.eMessageVerbose)
      THEN
        _stMsg.eType          := E_MessageType.eMessageVerbose;
        _stMsg.eSubdevice     := e_Subdevice.fbPower;
        _stMsg.iErrorNumber   := _nErrorId;
        _stMsg.sText          := concat('Axis Enable: ', TO_STRING(_eState));
        f_MessageSet(_stMsg);
      END_IF
    END_IF
END_CASE
//-----------------------------------------------------------------------------
//-----------------------------------------------------------------------------

Enable                   := _eState;
END_METHOD

METHOD GearIn : E_PROGRESS;
VAR_INPUT
  Execute             : BOOL;
  stMoveData          : ST_MOVE_DATA;
  stGearData          : ST_GEAR_DATA;
END_VAR
VAR_INST
  _nErrorId           : UDINT;
  _eState             : E_PROGRESS;
END_VAR
IF NOT Execute THEN _eState  := E_PROGRESS.PROGRESS_INIT; END_IF 
IF NOT Check() THEN GearIn   := E_PROGRESS.PROGRESS_ERROR; RETURN; END_IF


CASE _eState
OF
  E_PROGRESS.PROGRESS_INIT:
    IF Execute
    THEN
      _nErrorId               := 0;
      _eState                 := E_PROGRESS.PROGRESS_BUSY;

      IF NOT __ISVALIDREF(_Master)
      THEN
        _bError               := TRUE;
        _nErrorId             := 666;
        _eState               := E_PROGRESS.PROGRESS_ERROR;

        _stMsg.eType          := E_MessageType.eMessageError;
        _stMsg.eSubdevice     := e_Subdevice.fbGearIn;
        _stMsg.iErrorNumber   := _nErrorId;
        _stMsg.sText          := concat('Invalid Master Ref: ', TO_STRING(_eState));
        f_MessageSet(_stMsg);
      END_IF
    END_IF
END_CASE
//-----------------------------------------------------------------------------
//-----------------------------------------------------------------------------
CASE _eState
OF
  E_PROGRESS.PROGRESS_BUSY:
    _eState                   := E_PROGRESS.PROGRESS_PREPARE;
    _fbPower.Override         := stMoveData.rOverride;

    _fbGearIn(
            Master            := _Master, 
            Slave             := _Mover,
            Execute           := FALSE,
            RatioNumerator    := stGearData.rGearNumerator,
            RatioDenominator  := stGearData.iGearDenumerator, 
            Acceleration      := stMoveData.rAcc, 
            Deceleration      := stMoveData.rAcc, 
            Jerk              := stMoveData.rJerk, 
            BufferMode        := Tc2_MC2.MC_BufferMode.MC_Aborting);
END_CASE
//-----------------------------------------------------------------------------
//-----------------------------------------------------------------------------
CASE _eState
OF
  E_PROGRESS.PROGRESS_PREPARE:
    _fbGearIn(
            Master            := _Master, 
            Slave             := _Mover,
            Execute           := TRUE);

    IF _fbGearIn.Error
    THEN
      _bError                 := TRUE;
      _nErrorId               := _fbGearIn.ErrorID;
      _eState                 := E_PROGRESS.PROGRESS_ERROR;

      _stMsg.eType            := E_MessageType.eMessageError;
      _stMsg.eSubdevice       := e_Subdevice.fbGearIn;
      _stMsg.iErrorNumber     := _nErrorId;
      _stMsg.sText            := TO_STRING(_eState);
      f_MessageSet(_stMsg);

    ELSIF _fbGearIn.InGear
    THEN
      _eState                 := E_PROGRESS.PROGRESS_DONE;

